(* IEC 61131-3 sources: TIA2AX/tests/V19/test_projects/expected/HW_2200330/ST50_PLC, 7 files *)

(* ---- HwIdentifiers.st ---- *)
TYPE
	HwIdentifiers : WORD
	(
		ST50_PLC_Profilschiene_0 :=	WORD#256,
		ST50_PLC :=	WORD#48,
		ST50_PLC_Card_reader_writer_1 :=	WORD#51,
		ST50_PLC_CPU_display_1 :=	WORD#54,
		ST50_PLC_OPC_UA_1 :=	WORD#117,
		ST50_PLC_DP_interface_1 :=	WORD#60,
		ST50_PLC_PROFINET_interface_1 :=	WORD#64,
		ST50_PLC_PROFINET_interface_1_Port_1 :=	WORD#65,
		ST50_PLC_PROFINET_interface_1_Port_2 :=	WORD#66,
		ST50_PLC_PROFINET_interface_2 :=	WORD#72,
		ST50_PLC_PROFINET_interface_2_Port_1 :=	WORD#73,
		ST50_Switch_SCALANCE_X_rack :=	WORD#393,
		ST50_Switch :=	WORD#394,
		ST50_Switch_ST50_Switch :=	WORD#395,
		ST50_Switch_SCALANCE_interface_1 :=	WORD#396,
		ST50_Switch_SCALANCE_interface_1_Port_1 :=	WORD#397,
		ST50_Switch_SCALANCE_interface_1_Port_2 :=	WORD#398,
		ST50_Switch_SCALANCE_interface_1_Port_3 :=	WORD#399,
		ST50_Switch_SCALANCE_interface_1_Port_4 :=	WORD#400,
		ST50_Switch_SCALANCE_interface_1_Port_5 :=	WORD#401,
		ST50_Switch_SCALANCE_interface_1_Port_6 :=	WORD#402,
		ST50_Switch_SCALANCE_interface_1_Port_7 :=	WORD#403,
		ST50_Switch_SCALANCE_interface_1_Port_8 :=	WORD#404,
		ST50_Switch_SCALANCE_interface_1_Port_9 :=	WORD#405,
		ST50_Switch_SCALANCE_interface_1_Port_10 :=	WORD#406,
		ST50_Switch_SCALANCE_interface_1_Port_11 :=	WORD#407,
		ST50_Switch_SCALANCE_interface_1_Port_12 :=	WORD#408,
		ST50_Switch_SCALANCE_interface_1_Port_13 :=	WORD#409,
		ST50_Switch_SCALANCE_interface_1_Port_14 :=	WORD#410,
		ST50_Switch_SCALANCE_interface_1_Port_15 :=	WORD#411,
		ST50_Switch_SCALANCE_interface_1_Port_16 :=	WORD#412,
		ST50_Switch_1_SCALANCE_X_rack :=	WORD#416,
		ST50_Switch_1 :=	WORD#417,
		ST50_Switch_1_ST50_Switch_1 :=	WORD#418,
		ST50_Switch_1_SCALANCE_interface_1 :=	WORD#419,
		ST50_Switch_1_SCALANCE_interface_1_Port_1 :=	WORD#420,
		ST50_Switch_1_SCALANCE_interface_1_Port_2 :=	WORD#421,
		ST50_Switch_1_SCALANCE_interface_1_Port_3 :=	WORD#422,
		ST50_Switch_1_SCALANCE_interface_1_Port_4 :=	WORD#423,
		ST50_Switch_1_SCALANCE_interface_1_Port_5 :=	WORD#424,
		ST50_Switch_1_SCALANCE_interface_1_Port_6 :=	WORD#425,
		ST50_Switch_1_SCALANCE_interface_1_Port_7 :=	WORD#426,
		ST50_Switch_1_SCALANCE_interface_1_Port_8 :=	WORD#427,
		ST50_Switch_1_SCALANCE_interface_1_Port_9 :=	WORD#428,
		ST50_Switch_1_SCALANCE_interface_1_Port_10 :=	WORD#429,
		ST50_Switch_1_SCALANCE_interface_1_Port_11 :=	WORD#430,
		ST50_Switch_1_SCALANCE_interface_1_Port_12 :=	WORD#431,
		ST50_Switch_1_SCALANCE_interface_1_Port_13 :=	WORD#432,
		ST50_Switch_1_SCALANCE_interface_1_Port_14 :=	WORD#433,
		ST50_Switch_1_SCALANCE_interface_1_Port_15 :=	WORD#434,
		ST50_Switch_1_SCALANCE_interface_1_Port_16 :=	WORD#435,
		ST50_CPX_PN_IO_Interface :=	WORD#259,
		ST50_CPX_PN_IO_Interface_Port_1 :=	WORD#260,
		ST50_CPX_PN_IO_Interface_Port_2 :=	WORD#261,
		ST50_CPX_CPX :=	WORD#262,
		ST50_CPX_MPA1S_VMPA1_FB_EMS_8_8DO_1 :=	WORD#263,
		ST50_CPX_MPA1S_VMPA1_FB_EMS_8_8DO_2 :=	WORD#264,
		ST50_CPX_MPA1S_VMPA1_FB_EMS_8_8DO_3 :=	WORD#265,
		ST50_CPX_MPA1S_VMPA1_FB_EMS_8_8DO_4 :=	WORD#266,
		ST50_CPX_MPA1S_VMPA1_FB_EMS_8_8DO_5 :=	WORD#267,
		ST50_CPX_MPA1S_VMPA1_FB_EMS_8_8DO_6 :=	WORD#268,
		ST50_CPX_MPA1S_VMPA1_FB_EMS_8_8DO_7 :=	WORD#269,
		ST50_CPX_MPA1S_VMPA1_FB_EMS_8_8DO_8 :=	WORD#270,
		ST50_CPX_MPA1S_VMPA1_FB_EMS_8_8DO_9 :=	WORD#271,
		ST50_CPX_MPA1G_VMPA1_FB_EMG_8_8DO_6 :=	WORD#272,
		ST50_ET200SP_Rack_0 :=	WORD#277,
		ST50_ET200SP :=	WORD#278,
		ST50_ET200SP_ST50_ET200SP :=	WORD#279,
		ST50_ET200SP_PROFINET_interface :=	WORD#280,
		ST50_ET200SP_PROFINET_interface_Port_1 :=	WORD#282,
		ST50_ET200SP_PROFINET_interface_Port_2 :=	WORD#281,
		ST50_ET200SP_BA_2xRJ45 :=	WORD#282,
		ST50_ET200SP_CM_4xIO_Link_1 :=	WORD#283,
		ST50_ET200SP_CM_4xIO_Link_2 :=	WORD#284,
		ST50_ET200SP_DI_16x24VDC_ST_1 :=	WORD#285,
		ST50_ET200SP_DI_16x24VDC_ST_2 :=	WORD#286,
		ST50_ET200SP_DI_8x24VDC_ST_4 :=	WORD#287,
		ST50_ET200SP_DI_8x24VDC_ST_3 :=	WORD#288,
		ST50_ET200SP_DQ_16x24VDC_0_5A_ST_1 :=	WORD#289,
		ST50_ET200SP_DQ_16x24VDC_0_5A_ST_2 :=	WORD#290,
		ST50_ET200SP_DQ_16x24VDC_0_5A_ST_3 :=	WORD#291,
		ST50_ET200SP_Servermodul_1 :=	WORD#292,
		ST50_HMI_ConnectionBox_Connection_Box :=	WORD#294,
		ST50_HMI_ConnectionBox :=	WORD#295,
		ST50_HMI_ConnectionBox_ST50_HMI_ConnectionBox :=	WORD#296,
		ST50_HMI_ConnectionBox_SCALANCE_interface_1 :=	WORD#297,
		ST50_HMI_ConnectionBox_SCALANCE_interface_1_Port_1 :=	WORD#298,
		ST50_HMI_ConnectionBox_SCALANCE_interface_1_Port_2 :=	WORD#299,
		ST50_HMI_ConnectionBox_SCALANCE_interface_1_Port_3 :=	WORD#300,
		ST50_SCHUNK_L_Rack :=	WORD#302,
		ST50_SCHUNK_L :=	WORD#303,
		ST50_SCHUNK_L_Interface :=	WORD#304,
		ST50_SCHUNK_L_Interface_Port_1 :=	WORD#305,
		ST50_SCHUNK_L_Interface_Port_2 :=	WORD#306,
		ST50_SCHUNK_L_DEVICE_SFP :=	WORD#307,
		ST50_SCHUNK_L_IN_4_Double_Words :=	WORD#308,
		ST50_SCHUNK_L_OUT_4_Double_Words :=	WORD#309,
		ST50_SCHUNK_R_Rack :=	WORD#311,
		ST50_SCHUNK_R :=	WORD#312,
		ST50_SCHUNK_R_Interface :=	WORD#313,
		ST50_SCHUNK_R_Interface_Port_1 :=	WORD#314,
		ST50_SCHUNK_R_Interface_Port_2 :=	WORD#315,
		ST50_SCHUNK_R_DEVICE_SFP :=	WORD#316,
		ST50_SCHUNK_R_IN_4_Double_Words :=	WORD#317,
		ST50_SCHUNK_R_OUT_4_Double_Words :=	WORD#318,
		ST50_TZ535_PN_Rack :=	WORD#320,
		ST50_TZ535_PN :=	WORD#321,
		ST50_TZ535_PN_Interface :=	WORD#322,
		ST50_TZ535_PN_Interface_Port_1 :=	WORD#323,
		ST50_TZ535_PN_Interface_Port_2 :=	WORD#324,
		ST50_TZ535_PN_2D_TZ535_PN_PROFINET_IO :=	WORD#325,
		ST50_TZ535_PN_In_Out_32_byte_x :=	WORD#326,
		ST50_1_DM260_WPC_Rack :=	WORD#328,
		ST50_1_DM260_WPC :=	WORD#329,
		ST50_1_DM260_WPC_Interface :=	WORD#330,
		ST50_1_DM260_WPC_Interface_Port_1 :=	WORD#331,
		ST50_1_DM260_WPC_DataMan_260 :=	WORD#332,
		ST50_1_DM260_WPC_Acquisition_Control :=	WORD#333,
		ST50_1_DM260_WPC_Acquisition_Status :=	WORD#334,
		ST50_1_DM260_WPC_Results_Control :=	WORD#335,
		ST50_1_DM260_WPC_Results_Status :=	WORD#336,
		ST50_1_DM260_WPC_Soft_Event_Control :=	WORD#337,
		ST50_1_DM260_WPC_User_Data_64_bytes :=	WORD#338,
		ST50_1_DM260_WPC_Result_Data_64_bytes :=	WORD#339,
		ST50_1_DM260_Rack :=	WORD#341,
		ST50_1_DM260 :=	WORD#342,
		ST50_1_DM260_Interface :=	WORD#343,
		ST50_1_DM260_Interface_Port_1 :=	WORD#344,
		ST50_1_DM260_DataMan_260 :=	WORD#345,
		ST50_1_DM260_Acquisition_Control :=	WORD#346,
		ST50_1_DM260_Acquisition_Status :=	WORD#347,
		ST50_1_DM260_Results_Control :=	WORD#348,
		ST50_1_DM260_Results_Status :=	WORD#349,
		ST50_1_DM260_Soft_Event_Control :=	WORD#350,
		ST50_1_DM260_User_Data_64_bytes :=	WORD#351,
		ST50_1_DM260_Result_Data_64_bytes :=	WORD#352,
		ST50_2_DM260_Rack :=	WORD#354,
		ST50_2_DM260 :=	WORD#355,
		ST50_2_DM260_Interface :=	WORD#356,
		ST50_2_DM260_Interface_Port_1 :=	WORD#357,
		ST50_2_DM260_DataMan_260 :=	WORD#358,
		ST50_2_DM260_Acquisition_Control :=	WORD#359,
		ST50_2_DM260_Acquisition_Status :=	WORD#360,
		ST50_2_DM260_Results_Control :=	WORD#361,
		ST50_2_DM260_Results_Status :=	WORD#362,
		ST50_2_DM260_Soft_Event_Control :=	WORD#363,
		ST50_2_DM260_User_Data_64_bytes :=	WORD#364,
		ST50_2_DM260_Result_Data_64_bytes :=	WORD#365,
		ST50_3_DM260_Rack :=	WORD#367,
		ST50_3_DM260 :=	WORD#368,
		ST50_3_DM260_Interface :=	WORD#369,
		ST50_3_DM260_Interface_Port_1 :=	WORD#370,
		ST50_3_DM260_DataMan_260 :=	WORD#371,
		ST50_3_DM260_Acquisition_Control :=	WORD#372,
		ST50_3_DM260_Acquisition_Status :=	WORD#373,
		ST50_3_DM260_Results_Control :=	WORD#374,
		ST50_3_DM260_Results_Status :=	WORD#375,
		ST50_3_DM260_Soft_Event_Control :=	WORD#376,
		ST50_3_DM260_User_Data_64_bytes :=	WORD#377,
		ST50_3_DM260_Result_Data_64_bytes :=	WORD#378,
		ST50_4_DM260_Rack :=	WORD#380,
		ST50_4_DM260 :=	WORD#381,
		ST50_4_DM260_Interface :=	WORD#382,
		ST50_4_DM260_Interface_Port_1 :=	WORD#383,
		ST50_4_DM260_DataMan_260 :=	WORD#384,
		ST50_4_DM260_Acquisition_Control :=	WORD#385,
		ST50_4_DM260_Acquisition_Status :=	WORD#386,
		ST50_4_DM260_Results_Control :=	WORD#387,
		ST50_4_DM260_Results_Status :=	WORD#388,
		ST50_4_DM260_Soft_Event_Control :=	WORD#389,
		ST50_4_DM260_User_Data_64_bytes :=	WORD#390,
		ST50_4_DM260_Result_Data_64_bytes :=	WORD#391,
		NONE:= WORD#0
	);
END_TYPE

(* ---- HwInputs.st ---- *)
TYPE
	HwInputs : STRUCT
		ST50_ET200SP_CM_4xIO_Link_1 AT %B100 : ARRAY[0..31] OF BYTE;
		ST50_ET200SP_CM_4xIO_Link_2 AT %B132 : ARRAY[0..31] OF BYTE;
		ST50_ET200SP_DI_16x24VDC_ST_1 AT %B0 : WORD;
		ST50_ET200SP_DI_16x24VDC_ST_2 AT %B2 : WORD;
		ST50_ET200SP_DI_8x24VDC_ST_4 AT %B4 : BYTE;
		ST50_ET200SP_DI_8x24VDC_ST_3 AT %B5 : BYTE;
		ST50_SCHUNK_L_IN_4_Double_Words AT %B600 : ARRAY[0..15] OF BYTE;
		ST50_SCHUNK_R_IN_4_Double_Words AT %B616 : ARRAY[0..15] OF BYTE;
		ST50_TZ535_PN_In_Out_32_byte_x AT %B1000 : ARRAY[0..31] OF BYTE;
		ST50_1_DM260_WPC_Acquisition_Status AT %B3505 : ARRAY[0..2] OF BYTE;
		ST50_1_DM260_WPC_Results_Status AT %B3508 : BYTE;
		ST50_1_DM260_WPC_Soft_Event_Control AT %B3509 : BYTE;
		ST50_1_DM260_WPC_Result_Data_64_bytes AT %B3582 : ARRAY[0..71] OF BYTE;
		ST50_1_DM260_Acquisition_Status AT %B3654 : ARRAY[0..2] OF BYTE;
		ST50_1_DM260_Results_Status AT %B3657 : BYTE;
		ST50_1_DM260_Soft_Event_Control AT %B3658 : BYTE;
		ST50_1_DM260_Result_Data_64_bytes AT %B3659 : ARRAY[0..71] OF BYTE;
		ST50_2_DM260_Acquisition_Status AT %B3731 : ARRAY[0..2] OF BYTE;
		ST50_2_DM260_Results_Status AT %B3734 : BYTE;
		ST50_2_DM260_Soft_Event_Control AT %B3735 : BYTE;
		ST50_2_DM260_Result_Data_64_bytes AT %B3736 : ARRAY[0..71] OF BYTE;
		ST50_3_DM260_Acquisition_Status AT %B3808 : ARRAY[0..2] OF BYTE;
		ST50_3_DM260_Results_Status AT %B3811 : BYTE;
		ST50_3_DM260_Soft_Event_Control AT %B3812 : BYTE;
		ST50_3_DM260_Result_Data_64_bytes AT %B3813 : ARRAY[0..71] OF BYTE;
		ST50_4_DM260_Acquisition_Status AT %B3885 : ARRAY[0..2] OF BYTE;
		ST50_4_DM260_Results_Status AT %B3888 : BYTE;
		ST50_4_DM260_Soft_Event_Control AT %B3889 : BYTE;
		ST50_4_DM260_Result_Data_64_bytes AT %B3890 : ARRAY[0..71] OF BYTE;
	END_STRUCT;
END_TYPE

(* ---- HwOutputs.st ---- *)
TYPE
	HwOutputs : STRUCT
		ST50_CPX_MPA1S_VMPA1_FB_EMS_8_8DO_1 AT %B200 : BYTE;
		ST50_CPX_MPA1S_VMPA1_FB_EMS_8_8DO_2 AT %B201 : BYTE;
		ST50_CPX_MPA1S_VMPA1_FB_EMS_8_8DO_3 AT %B202 : BYTE;
		ST50_CPX_MPA1S_VMPA1_FB_EMS_8_8DO_4 AT %B203 : BYTE;
		ST50_CPX_MPA1S_VMPA1_FB_EMS_8_8DO_5 AT %B204 : BYTE;
		ST50_CPX_MPA1S_VMPA1_FB_EMS_8_8DO_6 AT %B205 : BYTE;
		ST50_CPX_MPA1S_VMPA1_FB_EMS_8_8DO_7 AT %B206 : BYTE;
		ST50_CPX_MPA1S_VMPA1_FB_EMS_8_8DO_8 AT %B207 : BYTE;
		ST50_CPX_MPA1S_VMPA1_FB_EMS_8_8DO_9 AT %B208 : BYTE;
		ST50_CPX_MPA1G_VMPA1_FB_EMG_8_8DO_6 AT %B209 : BYTE;
		ST50_ET200SP_CM_4xIO_Link_1 AT %B100 : ARRAY[0..31] OF BYTE;
		ST50_ET200SP_CM_4xIO_Link_2 AT %B132 : ARRAY[0..31] OF BYTE;
		ST50_ET200SP_DQ_16x24VDC_0_5A_ST_1 AT %B0 : WORD;
		ST50_ET200SP_DQ_16x24VDC_0_5A_ST_2 AT %B2 : WORD;
		ST50_ET200SP_DQ_16x24VDC_0_5A_ST_3 AT %B4 : WORD;
		ST50_SCHUNK_L_OUT_4_Double_Words AT %B600 : ARRAY[0..15] OF BYTE;
		ST50_SCHUNK_R_OUT_4_Double_Words AT %B616 : ARRAY[0..15] OF BYTE;
		ST50_TZ535_PN_In_Out_32_byte_x AT %B1000 : ARRAY[0..31] OF BYTE;
		ST50_1_DM260_WPC_Acquisition_Control AT %B3501 : BYTE;
		ST50_1_DM260_WPC_Results_Control AT %B3505 : BYTE;
		ST50_1_DM260_WPC_Soft_Event_Control AT %B3506 : BYTE;
		ST50_1_DM260_WPC_User_Data_64_bytes AT %B3578 : ARRAY[0..67] OF BYTE;
		ST50_1_DM260_Acquisition_Control AT %B3502 : BYTE;
		ST50_1_DM260_Results_Control AT %B3507 : BYTE;
		ST50_1_DM260_Soft_Event_Control AT %B3508 : BYTE;
		ST50_1_DM260_User_Data_64_bytes AT %B3646 : ARRAY[0..67] OF BYTE;
		ST50_2_DM260_Acquisition_Control AT %B3509 : BYTE;
		ST50_2_DM260_Results_Control AT %B3714 : BYTE;
		ST50_2_DM260_Soft_Event_Control AT %B3715 : BYTE;
		ST50_2_DM260_User_Data_64_bytes AT %B3716 : ARRAY[0..67] OF BYTE;
		ST50_3_DM260_Acquisition_Control AT %B3784 : BYTE;
		ST50_3_DM260_Results_Control AT %B3785 : BYTE;
		ST50_3_DM260_Soft_Event_Control AT %B3786 : BYTE;
		ST50_3_DM260_User_Data_64_bytes AT %B3787 : ARRAY[0..67] OF BYTE;
		ST50_4_DM260_Acquisition_Control AT %B3855 : BYTE;
		ST50_4_DM260_Results_Control AT %B3856 : BYTE;
		ST50_4_DM260_Soft_Event_Control AT %B3857 : BYTE;
		ST50_4_DM260_User_Data_64_bytes AT %B3858 : ARRAY[0..67] OF BYTE;
	END_STRUCT;
END_TYPE

(* ---- PlcInputs.st ---- *)
TYPE
	PlcInputs : STRUCT
		ST50_ET200SP_CM_4xIO_Link_1 : ARRAY[0..31] OF BYTE;
		ST50_ET200SP_CM_4xIO_Link_2 : ARRAY[0..31] OF BYTE;
		ST50_ET200SP_DI_16x24VDC_ST_1 : WORD;
		ST50_ET200SP_DI_16x24VDC_ST_2 : WORD;
		ST50_ET200SP_DI_8x24VDC_ST_4 : BYTE;
		ST50_ET200SP_DI_8x24VDC_ST_3 : BYTE;
		ST50_SCHUNK_L_IN_4_Double_Words : ARRAY[0..15] OF BYTE;
		ST50_SCHUNK_R_IN_4_Double_Words : ARRAY[0..15] OF BYTE;
		ST50_TZ535_PN_In_Out_32_byte_x : ARRAY[0..31] OF BYTE;
		ST50_1_DM260_WPC_Acquisition_Status : ARRAY[0..2] OF BYTE;
		ST50_1_DM260_WPC_Results_Status : BYTE;
		ST50_1_DM260_WPC_Soft_Event_Control : BYTE;
		ST50_1_DM260_WPC_Result_Data_64_bytes : ARRAY[0..71] OF BYTE;
		ST50_1_DM260_Acquisition_Status : ARRAY[0..2] OF BYTE;
		ST50_1_DM260_Results_Status : BYTE;
		ST50_1_DM260_Soft_Event_Control : BYTE;
		ST50_1_DM260_Result_Data_64_bytes : ARRAY[0..71] OF BYTE;
		ST50_2_DM260_Acquisition_Status : ARRAY[0..2] OF BYTE;
		ST50_2_DM260_Results_Status : BYTE;
		ST50_2_DM260_Soft_Event_Control : BYTE;
		ST50_2_DM260_Result_Data_64_bytes : ARRAY[0..71] OF BYTE;
		ST50_3_DM260_Acquisition_Status : ARRAY[0..2] OF BYTE;
		ST50_3_DM260_Results_Status : BYTE;
		ST50_3_DM260_Soft_Event_Control : BYTE;
		ST50_3_DM260_Result_Data_64_bytes : ARRAY[0..71] OF BYTE;
		ST50_4_DM260_Acquisition_Status : ARRAY[0..2] OF BYTE;
		ST50_4_DM260_Results_Status : BYTE;
		ST50_4_DM260_Soft_Event_Control : BYTE;
		ST50_4_DM260_Result_Data_64_bytes : ARRAY[0..71] OF BYTE;
	END_STRUCT;
END_TYPE

(* ---- PlcOutputs.st ---- *)
TYPE
	PlcOutputs : STRUCT
		ST50_CPX_MPA1S_VMPA1_FB_EMS_8_8DO_1 : BYTE;
		ST50_CPX_MPA1S_VMPA1_FB_EMS_8_8DO_2 : BYTE;
		ST50_CPX_MPA1S_VMPA1_FB_EMS_8_8DO_3 : BYTE;
		ST50_CPX_MPA1S_VMPA1_FB_EMS_8_8DO_4 : BYTE;
		ST50_CPX_MPA1S_VMPA1_FB_EMS_8_8DO_5 : BYTE;
		ST50_CPX_MPA1S_VMPA1_FB_EMS_8_8DO_6 : BYTE;
		ST50_CPX_MPA1S_VMPA1_FB_EMS_8_8DO_7 : BYTE;
		ST50_CPX_MPA1S_VMPA1_FB_EMS_8_8DO_8 : BYTE;
		ST50_CPX_MPA1S_VMPA1_FB_EMS_8_8DO_9 : BYTE;
		ST50_CPX_MPA1G_VMPA1_FB_EMG_8_8DO_6 : BYTE;
		ST50_ET200SP_CM_4xIO_Link_1 : ARRAY[0..31] OF BYTE;
		ST50_ET200SP_CM_4xIO_Link_2 : ARRAY[0..31] OF BYTE;
		ST50_ET200SP_DQ_16x24VDC_0_5A_ST_1 : WORD;
		ST50_ET200SP_DQ_16x24VDC_0_5A_ST_2 : WORD;
		ST50_ET200SP_DQ_16x24VDC_0_5A_ST_3 : WORD;
		ST50_SCHUNK_L_OUT_4_Double_Words : ARRAY[0..15] OF BYTE;
		ST50_SCHUNK_R_OUT_4_Double_Words : ARRAY[0..15] OF BYTE;
		ST50_TZ535_PN_In_Out_32_byte_x : ARRAY[0..31] OF BYTE;
		ST50_1_DM260_WPC_Acquisition_Control : BYTE;
		ST50_1_DM260_WPC_Results_Control : BYTE;
		ST50_1_DM260_WPC_Soft_Event_Control : BYTE;
		ST50_1_DM260_WPC_User_Data_64_bytes : ARRAY[0..67] OF BYTE;
		ST50_1_DM260_Acquisition_Control : BYTE;
		ST50_1_DM260_Results_Control : BYTE;
		ST50_1_DM260_Soft_Event_Control : BYTE;
		ST50_1_DM260_User_Data_64_bytes : ARRAY[0..67] OF BYTE;
		ST50_2_DM260_Acquisition_Control : BYTE;
		ST50_2_DM260_Results_Control : BYTE;
		ST50_2_DM260_Soft_Event_Control : BYTE;
		ST50_2_DM260_User_Data_64_bytes : ARRAY[0..67] OF BYTE;
		ST50_3_DM260_Acquisition_Control : BYTE;
		ST50_3_DM260_Results_Control : BYTE;
		ST50_3_DM260_Soft_Event_Control : BYTE;
		ST50_3_DM260_User_Data_64_bytes : ARRAY[0..67] OF BYTE;
		ST50_4_DM260_Acquisition_Control : BYTE;
		ST50_4_DM260_Results_Control : BYTE;
		ST50_4_DM260_Soft_Event_Control : BYTE;
		ST50_4_DM260_User_Data_64_bytes : ARRAY[0..67] OF BYTE;
	END_STRUCT;
END_TYPE

(* ---- CopyInputs.st ---- *)
FUNCTION CopyInputs
	VAR_EXTERNAL
		HwInputs : HwInputs;
		PlcInputs : PlcInputs;
	END_VAR
	PlcInputs.ST50_ET200SP_CM_4xIO_Link_1[0] := HwInputs.ST50_ET200SP_CM_4xIO_Link_1[0];
	PlcInputs.ST50_ET200SP_CM_4xIO_Link_1[1] := HwInputs.ST50_ET200SP_CM_4xIO_Link_1[1];
	PlcInputs.ST50_ET200SP_CM_4xIO_Link_1[2] := HwInputs.ST50_ET200SP_CM_4xIO_Link_1[2];
	PlcInputs.ST50_ET200SP_CM_4xIO_Link_1[3] := HwInputs.ST50_ET200SP_CM_4xIO_Link_1[3];
	PlcInputs.ST50_ET200SP_CM_4xIO_Link_1[4] := HwInputs.ST50_ET200SP_CM_4xIO_Link_1[4];
	PlcInputs.ST50_ET200SP_CM_4xIO_Link_1[5] := HwInputs.ST50_ET200SP_CM_4xIO_Link_1[5];
	PlcInputs.ST50_ET200SP_CM_4xIO_Link_1[6] := HwInputs.ST50_ET200SP_CM_4xIO_Link_1[6];
	PlcInputs.ST50_ET200SP_CM_4xIO_Link_1[7] := HwInputs.ST50_ET200SP_CM_4xIO_Link_1[7];
	PlcInputs.ST50_ET200SP_CM_4xIO_Link_1[8] := HwInputs.ST50_ET200SP_CM_4xIO_Link_1[8];
	PlcInputs.ST50_ET200SP_CM_4xIO_Link_1[9] := HwInputs.ST50_ET200SP_CM_4xIO_Link_1[9];
	PlcInputs.ST50_ET200SP_CM_4xIO_Link_1[10] := HwInputs.ST50_ET200SP_CM_4xIO_Link_1[10];
	PlcInputs.ST50_ET200SP_CM_4xIO_Link_1[11] := HwInputs.ST50_ET200SP_CM_4xIO_Link_1[11];
	PlcInputs.ST50_ET200SP_CM_4xIO_Link_1[12] := HwInputs.ST50_ET200SP_CM_4xIO_Link_1[12];
	PlcInputs.ST50_ET200SP_CM_4xIO_Link_1[13] := HwInputs.ST50_ET200SP_CM_4xIO_Link_1[13];
	PlcInputs.ST50_ET200SP_CM_4xIO_Link_1[14] := HwInputs.ST50_ET200SP_CM_4xIO_Link_1[14];
	PlcInputs.ST50_ET200SP_CM_4xIO_Link_1[15] := HwInputs.ST50_ET200SP_CM_4xIO_Link_1[15];
	PlcInputs.ST50_ET200SP_CM_4xIO_Link_1[16] := HwInputs.ST50_ET200SP_CM_4xIO_Link_1[16];
	PlcInputs.ST50_ET200SP_CM_4xIO_Link_1[17] := HwInputs.ST50_ET200SP_CM_4xIO_Link_1[17];
	PlcInputs.ST50_ET200SP_CM_4xIO_Link_1[18] := HwInputs.ST50_ET200SP_CM_4xIO_Link_1[18];
	PlcInputs.ST50_ET200SP_CM_4xIO_Link_1[19] := HwInputs.ST50_ET200SP_CM_4xIO_Link_1[19];
	PlcInputs.ST50_ET200SP_CM_4xIO_Link_1[20] := HwInputs.ST50_ET200SP_CM_4xIO_Link_1[20];
	PlcInputs.ST50_ET200SP_CM_4xIO_Link_1[21] := HwInputs.ST50_ET200SP_CM_4xIO_Link_1[21];
	PlcInputs.ST50_ET200SP_CM_4xIO_Link_1[22] := HwInputs.ST50_ET200SP_CM_4xIO_Link_1[22];
	PlcInputs.ST50_ET200SP_CM_4xIO_Link_1[23] := HwInputs.ST50_ET200SP_CM_4xIO_Link_1[23];
	PlcInputs.ST50_ET200SP_CM_4xIO_Link_1[24] := HwInputs.ST50_ET200SP_CM_4xIO_Link_1[24];
	PlcInputs.ST50_ET200SP_CM_4xIO_Link_1[25] := HwInputs.ST50_ET200SP_CM_4xIO_Link_1[25];
	PlcInputs.ST50_ET200SP_CM_4xIO_Link_1[26] := HwInputs.ST50_ET200SP_CM_4xIO_Link_1[26];
	PlcInputs.ST50_ET200SP_CM_4xIO_Link_1[27] := HwInputs.ST50_ET200SP_CM_4xIO_Link_1[27];
	PlcInputs.ST50_ET200SP_CM_4xIO_Link_1[28] := HwInputs.ST50_ET200SP_CM_4xIO_Link_1[28];
	PlcInputs.ST50_ET200SP_CM_4xIO_Link_1[29] := HwInputs.ST50_ET200SP_CM_4xIO_Link_1[29];
	PlcInputs.ST50_ET200SP_CM_4xIO_Link_1[30] := HwInputs.ST50_ET200SP_CM_4xIO_Link_1[30];
	PlcInputs.ST50_ET200SP_CM_4xIO_Link_1[31] := HwInputs.ST50_ET200SP_CM_4xIO_Link_1[31];
	PlcInputs.ST50_ET200SP_CM_4xIO_Link_2[0] := HwInputs.ST50_ET200SP_CM_4xIO_Link_2[0];
	PlcInputs.ST50_ET200SP_CM_4xIO_Link_2[1] := HwInputs.ST50_ET200SP_CM_4xIO_Link_2[1];
	PlcInputs.ST50_ET200SP_CM_4xIO_Link_2[2] := HwInputs.ST50_ET200SP_CM_4xIO_Link_2[2];
	PlcInputs.ST50_ET200SP_CM_4xIO_Link_2[3] := HwInputs.ST50_ET200SP_CM_4xIO_Link_2[3];
	PlcInputs.ST50_ET200SP_CM_4xIO_Link_2[4] := HwInputs.ST50_ET200SP_CM_4xIO_Link_2[4];
	PlcInputs.ST50_ET200SP_CM_4xIO_Link_2[5] := HwInputs.ST50_ET200SP_CM_4xIO_Link_2[5];
	PlcInputs.ST50_ET200SP_CM_4xIO_Link_2[6] := HwInputs.ST50_ET200SP_CM_4xIO_Link_2[6];
	PlcInputs.ST50_ET200SP_CM_4xIO_Link_2[7] := HwInputs.ST50_ET200SP_CM_4xIO_Link_2[7];
	PlcInputs.ST50_ET200SP_CM_4xIO_Link_2[8] := HwInputs.ST50_ET200SP_CM_4xIO_Link_2[8];
	PlcInputs.ST50_ET200SP_CM_4xIO_Link_2[9] := HwInputs.ST50_ET200SP_CM_4xIO_Link_2[9];
	PlcInputs.ST50_ET200SP_CM_4xIO_Link_2[10] := HwInputs.ST50_ET200SP_CM_4xIO_Link_2[10];
	PlcInputs.ST50_ET200SP_CM_4xIO_Link_2[11] := HwInputs.ST50_ET200SP_CM_4xIO_Link_2[11];
	PlcInputs.ST50_ET200SP_CM_4xIO_Link_2[12] := HwInputs.ST50_ET200SP_CM_4xIO_Link_2[12];
	PlcInputs.ST50_ET200SP_CM_4xIO_Link_2[13] := HwInputs.ST50_ET200SP_CM_4xIO_Link_2[13];
	PlcInputs.ST50_ET200SP_CM_4xIO_Link_2[14] := HwInputs.ST50_ET200SP_CM_4xIO_Link_2[14];
	PlcInputs.ST50_ET200SP_CM_4xIO_Link_2[15] := HwInputs.ST50_ET200SP_CM_4xIO_Link_2[15];
	PlcInputs.ST50_ET200SP_CM_4xIO_Link_2[16] := HwInputs.ST50_ET200SP_CM_4xIO_Link_2[16];
	PlcInputs.ST50_ET200SP_CM_4xIO_Link_2[17] := HwInputs.ST50_ET200SP_CM_4xIO_Link_2[17];
	PlcInputs.ST50_ET200SP_CM_4xIO_Link_2[18] := HwInputs.ST50_ET200SP_CM_4xIO_Link_2[18];
	PlcInputs.ST50_ET200SP_CM_4xIO_Link_2[19] := HwInputs.ST50_ET200SP_CM_4xIO_Link_2[19];
	PlcInputs.ST50_ET200SP_CM_4xIO_Link_2[20] := HwInputs.ST50_ET200SP_CM_4xIO_Link_2[20];
	PlcInputs.ST50_ET200SP_CM_4xIO_Link_2[21] := HwInputs.ST50_ET200SP_CM_4xIO_Link_2[21];
	PlcInputs.ST50_ET200SP_CM_4xIO_Link_2[22] := HwInputs.ST50_ET200SP_CM_4xIO_Link_2[22];
	PlcInputs.ST50_ET200SP_CM_4xIO_Link_2[23] := HwInputs.ST50_ET200SP_CM_4xIO_Link_2[23];
	PlcInputs.ST50_ET200SP_CM_4xIO_Link_2[24] := HwInputs.ST50_ET200SP_CM_4xIO_Link_2[24];
	PlcInputs.ST50_ET200SP_CM_4xIO_Link_2[25] := HwInputs.ST50_ET200SP_CM_4xIO_Link_2[25];
	PlcInputs.ST50_ET200SP_CM_4xIO_Link_2[26] := HwInputs.ST50_ET200SP_CM_4xIO_Link_2[26];
	PlcInputs.ST50_ET200SP_CM_4xIO_Link_2[27] := HwInputs.ST50_ET200SP_CM_4xIO_Link_2[27];
	PlcInputs.ST50_ET200SP_CM_4xIO_Link_2[28] := HwInputs.ST50_ET200SP_CM_4xIO_Link_2[28];
	PlcInputs.ST50_ET200SP_CM_4xIO_Link_2[29] := HwInputs.ST50_ET200SP_CM_4xIO_Link_2[29];
	PlcInputs.ST50_ET200SP_CM_4xIO_Link_2[30] := HwInputs.ST50_ET200SP_CM_4xIO_Link_2[30];
	PlcInputs.ST50_ET200SP_CM_4xIO_Link_2[31] := HwInputs.ST50_ET200SP_CM_4xIO_Link_2[31];
	PlcInputs.ST50_ET200SP_DI_16x24VDC_ST_1 := HwInputs.ST50_ET200SP_DI_16x24VDC_ST_1;
	PlcInputs.ST50_ET200SP_DI_16x24VDC_ST_2 := HwInputs.ST50_ET200SP_DI_16x24VDC_ST_2;
	PlcInputs.ST50_ET200SP_DI_8x24VDC_ST_4 := HwInputs.ST50_ET200SP_DI_8x24VDC_ST_4;
	PlcInputs.ST50_ET200SP_DI_8x24VDC_ST_3 := HwInputs.ST50_ET200SP_DI_8x24VDC_ST_3;
	PlcInputs.ST50_SCHUNK_L_IN_4_Double_Words[0] := HwInputs.ST50_SCHUNK_L_IN_4_Double_Words[0];
	PlcInputs.ST50_SCHUNK_L_IN_4_Double_Words[1] := HwInputs.ST50_SCHUNK_L_IN_4_Double_Words[1];
	PlcInputs.ST50_SCHUNK_L_IN_4_Double_Words[2] := HwInputs.ST50_SCHUNK_L_IN_4_Double_Words[2];
	PlcInputs.ST50_SCHUNK_L_IN_4_Double_Words[3] := HwInputs.ST50_SCHUNK_L_IN_4_Double_Words[3];
	PlcInputs.ST50_SCHUNK_L_IN_4_Double_Words[4] := HwInputs.ST50_SCHUNK_L_IN_4_Double_Words[4];
	PlcInputs.ST50_SCHUNK_L_IN_4_Double_Words[5] := HwInputs.ST50_SCHUNK_L_IN_4_Double_Words[5];
	PlcInputs.ST50_SCHUNK_L_IN_4_Double_Words[6] := HwInputs.ST50_SCHUNK_L_IN_4_Double_Words[6];
	PlcInputs.ST50_SCHUNK_L_IN_4_Double_Words[7] := HwInputs.ST50_SCHUNK_L_IN_4_Double_Words[7];
	PlcInputs.ST50_SCHUNK_L_IN_4_Double_Words[8] := HwInputs.ST50_SCHUNK_L_IN_4_Double_Words[8];
	PlcInputs.ST50_SCHUNK_L_IN_4_Double_Words[9] := HwInputs.ST50_SCHUNK_L_IN_4_Double_Words[9];
	PlcInputs.ST50_SCHUNK_L_IN_4_Double_Words[10] := HwInputs.ST50_SCHUNK_L_IN_4_Double_Words[10];
	PlcInputs.ST50_SCHUNK_L_IN_4_Double_Words[11] := HwInputs.ST50_SCHUNK_L_IN_4_Double_Words[11];
	PlcInputs.ST50_SCHUNK_L_IN_4_Double_Words[12] := HwInputs.ST50_SCHUNK_L_IN_4_Double_Words[12];
	PlcInputs.ST50_SCHUNK_L_IN_4_Double_Words[13] := HwInputs.ST50_SCHUNK_L_IN_4_Double_Words[13];
	PlcInputs.ST50_SCHUNK_L_IN_4_Double_Words[14] := HwInputs.ST50_SCHUNK_L_IN_4_Double_Words[14];
	PlcInputs.ST50_SCHUNK_L_IN_4_Double_Words[15] := HwInputs.ST50_SCHUNK_L_IN_4_Double_Words[15];
	PlcInputs.ST50_SCHUNK_R_IN_4_Double_Words[0] := HwInputs.ST50_SCHUNK_R_IN_4_Double_Words[0];
	PlcInputs.ST50_SCHUNK_R_IN_4_Double_Words[1] := HwInputs.ST50_SCHUNK_R_IN_4_Double_Words[1];
	PlcInputs.ST50_SCHUNK_R_IN_4_Double_Words[2] := HwInputs.ST50_SCHUNK_R_IN_4_Double_Words[2];
	PlcInputs.ST50_SCHUNK_R_IN_4_Double_Words[3] := HwInputs.ST50_SCHUNK_R_IN_4_Double_Words[3];
	PlcInputs.ST50_SCHUNK_R_IN_4_Double_Words[4] := HwInputs.ST50_SCHUNK_R_IN_4_Double_Words[4];
	PlcInputs.ST50_SCHUNK_R_IN_4_Double_Words[5] := HwInputs.ST50_SCHUNK_R_IN_4_Double_Words[5];
	PlcInputs.ST50_SCHUNK_R_IN_4_Double_Words[6] := HwInputs.ST50_SCHUNK_R_IN_4_Double_Words[6];
	PlcInputs.ST50_SCHUNK_R_IN_4_Double_Words[7] := HwInputs.ST50_SCHUNK_R_IN_4_Double_Words[7];
	PlcInputs.ST50_SCHUNK_R_IN_4_Double_Words[8] := HwInputs.ST50_SCHUNK_R_IN_4_Double_Words[8];
	PlcInputs.ST50_SCHUNK_R_IN_4_Double_Words[9] := HwInputs.ST50_SCHUNK_R_IN_4_Double_Words[9];
	PlcInputs.ST50_SCHUNK_R_IN_4_Double_Words[10] := HwInputs.ST50_SCHUNK_R_IN_4_Double_Words[10];
	PlcInputs.ST50_SCHUNK_R_IN_4_Double_Words[11] := HwInputs.ST50_SCHUNK_R_IN_4_Double_Words[11];
	PlcInputs.ST50_SCHUNK_R_IN_4_Double_Words[12] := HwInputs.ST50_SCHUNK_R_IN_4_Double_Words[12];
	PlcInputs.ST50_SCHUNK_R_IN_4_Double_Words[13] := HwInputs.ST50_SCHUNK_R_IN_4_Double_Words[13];
	PlcInputs.ST50_SCHUNK_R_IN_4_Double_Words[14] := HwInputs.ST50_SCHUNK_R_IN_4_Double_Words[14];
	PlcInputs.ST50_SCHUNK_R_IN_4_Double_Words[15] := HwInputs.ST50_SCHUNK_R_IN_4_Double_Words[15];
	PlcInputs.ST50_TZ535_PN_In_Out_32_byte_x[0] := HwInputs.ST50_TZ535_PN_In_Out_32_byte_x[0];
	PlcInputs.ST50_TZ535_PN_In_Out_32_byte_x[1] := HwInputs.ST50_TZ535_PN_In_Out_32_byte_x[1];
	PlcInputs.ST50_TZ535_PN_In_Out_32_byte_x[2] := HwInputs.ST50_TZ535_PN_In_Out_32_byte_x[2];
	PlcInputs.ST50_TZ535_PN_In_Out_32_byte_x[3] := HwInputs.ST50_TZ535_PN_In_Out_32_byte_x[3];
	PlcInputs.ST50_TZ535_PN_In_Out_32_byte_x[4] := HwInputs.ST50_TZ535_PN_In_Out_32_byte_x[4];
	PlcInputs.ST50_TZ535_PN_In_Out_32_byte_x[5] := HwInputs.ST50_TZ535_PN_In_Out_32_byte_x[5];
	PlcInputs.ST50_TZ535_PN_In_Out_32_byte_x[6] := HwInputs.ST50_TZ535_PN_In_Out_32_byte_x[6];
	PlcInputs.ST50_TZ535_PN_In_Out_32_byte_x[7] := HwInputs.ST50_TZ535_PN_In_Out_32_byte_x[7];
	PlcInputs.ST50_TZ535_PN_In_Out_32_byte_x[8] := HwInputs.ST50_TZ535_PN_In_Out_32_byte_x[8];
	PlcInputs.ST50_TZ535_PN_In_Out_32_byte_x[9] := HwInputs.ST50_TZ535_PN_In_Out_32_byte_x[9];
	PlcInputs.ST50_TZ535_PN_In_Out_32_byte_x[10] := HwInputs.ST50_TZ535_PN_In_Out_32_byte_x[10];
	PlcInputs.ST50_TZ535_PN_In_Out_32_byte_x[11] := HwInputs.ST50_TZ535_PN_In_Out_32_byte_x[11];
	PlcInputs.ST50_TZ535_PN_In_Out_32_byte_x[12] := HwInputs.ST50_TZ535_PN_In_Out_32_byte_x[12];
	PlcInputs.ST50_TZ535_PN_In_Out_32_byte_x[13] := HwInputs.ST50_TZ535_PN_In_Out_32_byte_x[13];
	PlcInputs.ST50_TZ535_PN_In_Out_32_byte_x[14] := HwInputs.ST50_TZ535_PN_In_Out_32_byte_x[14];
	PlcInputs.ST50_TZ535_PN_In_Out_32_byte_x[15] := HwInputs.ST50_TZ535_PN_In_Out_32_byte_x[15];
	PlcInputs.ST50_TZ535_PN_In_Out_32_byte_x[16] := HwInputs.ST50_TZ535_PN_In_Out_32_byte_x[16];
	PlcInputs.ST50_TZ535_PN_In_Out_32_byte_x[17] := HwInputs.ST50_TZ535_PN_In_Out_32_byte_x[17];
	PlcInputs.ST50_TZ535_PN_In_Out_32_byte_x[18] := HwInputs.ST50_TZ535_PN_In_Out_32_byte_x[18];
	PlcInputs.ST50_TZ535_PN_In_Out_32_byte_x[19] := HwInputs.ST50_TZ535_PN_In_Out_32_byte_x[19];
	PlcInputs.ST50_TZ535_PN_In_Out_32_byte_x[20] := HwInputs.ST50_TZ535_PN_In_Out_32_byte_x[20];
	PlcInputs.ST50_TZ535_PN_In_Out_32_byte_x[21] := HwInputs.ST50_TZ535_PN_In_Out_32_byte_x[21];
	PlcInputs.ST50_TZ535_PN_In_Out_32_byte_x[22] := HwInputs.ST50_TZ535_PN_In_Out_32_byte_x[22];
	PlcInputs.ST50_TZ535_PN_In_Out_32_byte_x[23] := HwInputs.ST50_TZ535_PN_In_Out_32_byte_x[23];
	PlcInputs.ST50_TZ535_PN_In_Out_32_byte_x[24] := HwInputs.ST50_TZ535_PN_In_Out_32_byte_x[24];
	PlcInputs.ST50_TZ535_PN_In_Out_32_byte_x[25] := HwInputs.ST50_TZ535_PN_In_Out_32_byte_x[25];
	PlcInputs.ST50_TZ535_PN_In_Out_32_byte_x[26] := HwInputs.ST50_TZ535_PN_In_Out_32_byte_x[26];
	PlcInputs.ST50_TZ535_PN_In_Out_32_byte_x[27] := HwInputs.ST50_TZ535_PN_In_Out_32_byte_x[27];
	PlcInputs.ST50_TZ535_PN_In_Out_32_byte_x[28] := HwInputs.ST50_TZ535_PN_In_Out_32_byte_x[28];
	PlcInputs.ST50_TZ535_PN_In_Out_32_byte_x[29] := HwInputs.ST50_TZ535_PN_In_Out_32_byte_x[29];
	PlcInputs.ST50_TZ535_PN_In_Out_32_byte_x[30] := HwInputs.ST50_TZ535_PN_In_Out_32_byte_x[30];
	PlcInputs.ST50_TZ535_PN_In_Out_32_byte_x[31] := HwInputs.ST50_TZ535_PN_In_Out_32_byte_x[31];
	PlcInputs.ST50_1_DM260_WPC_Acquisition_Status[0] := HwInputs.ST50_1_DM260_WPC_Acquisition_Status[0];
	PlcInputs.ST50_1_DM260_WPC_Acquisition_Status[1] := HwInputs.ST50_1_DM260_WPC_Acquisition_Status[1];
	PlcInputs.ST50_1_DM260_WPC_Acquisition_Status[2] := HwInputs.ST50_1_DM260_WPC_Acquisition_Status[2];
	PlcInputs.ST50_1_DM260_WPC_Results_Status := HwInputs.ST50_1_DM260_WPC_Results_Status;
	PlcInputs.ST50_1_DM260_WPC_Soft_Event_Control := HwInputs.ST50_1_DM260_WPC_Soft_Event_Control;
	PlcInputs.ST50_1_DM260_WPC_Result_Data_64_bytes[0] := HwInputs.ST50_1_DM260_WPC_Result_Data_64_bytes[0];
	PlcInputs.ST50_1_DM260_WPC_Result_Data_64_bytes[1] := HwInputs.ST50_1_DM260_WPC_Result_Data_64_bytes[1];
	PlcInputs.ST50_1_DM260_WPC_Result_Data_64_bytes[2] := HwInputs.ST50_1_DM260_WPC_Result_Data_64_bytes[2];
	PlcInputs.ST50_1_DM260_WPC_Result_Data_64_bytes[3] := HwInputs.ST50_1_DM260_WPC_Result_Data_64_bytes[3];
	PlcInputs.ST50_1_DM260_WPC_Result_Data_64_bytes[4] := HwInputs.ST50_1_DM260_WPC_Result_Data_64_bytes[4];
	PlcInputs.ST50_1_DM260_WPC_Result_Data_64_bytes[5] := HwInputs.ST50_1_DM260_WPC_Result_Data_64_bytes[5];
	PlcInputs.ST50_1_DM260_WPC_Result_Data_64_bytes[6] := HwInputs.ST50_1_DM260_WPC_Result_Data_64_bytes[6];
	PlcInputs.ST50_1_DM260_WPC_Result_Data_64_bytes[7] := HwInputs.ST50_1_DM260_WPC_Result_Data_64_bytes[7];
	PlcInputs.ST50_1_DM260_WPC_Result_Data_64_bytes[8] := HwInputs.ST50_1_DM260_WPC_Result_Data_64_bytes[8];
	PlcInputs.ST50_1_DM260_WPC_Result_Data_64_bytes[9] := HwInputs.ST50_1_DM260_WPC_Result_Data_64_bytes[9];
	PlcInputs.ST50_1_DM260_WPC_Result_Data_64_bytes[10] := HwInputs.ST50_1_DM260_WPC_Result_Data_64_bytes[10];
	PlcInputs.ST50_1_DM260_WPC_Result_Data_64_bytes[11] := HwInputs.ST50_1_DM260_WPC_Result_Data_64_bytes[11];
	PlcInputs.ST50_1_DM260_WPC_Result_Data_64_bytes[12] := HwInputs.ST50_1_DM260_WPC_Result_Data_64_bytes[12];
	PlcInputs.ST50_1_DM260_WPC_Result_Data_64_bytes[13] := HwInputs.ST50_1_DM260_WPC_Result_Data_64_bytes[13];
	PlcInputs.ST50_1_DM260_WPC_Result_Data_64_bytes[14] := HwInputs.ST50_1_DM260_WPC_Result_Data_64_bytes[14];
	PlcInputs.ST50_1_DM260_WPC_Result_Data_64_bytes[15] := HwInputs.ST50_1_DM260_WPC_Result_Data_64_bytes[15];
	PlcInputs.ST50_1_DM260_WPC_Result_Data_64_bytes[16] := HwInputs.ST50_1_DM260_WPC_Result_Data_64_bytes[16];
	PlcInputs.ST50_1_DM260_WPC_Result_Data_64_bytes[17] := HwInputs.ST50_1_DM260_WPC_Result_Data_64_bytes[17];
	PlcInputs.ST50_1_DM260_WPC_Result_Data_64_bytes[18] := HwInputs.ST50_1_DM260_WPC_Result_Data_64_bytes[18];
	PlcInputs.ST50_1_DM260_WPC_Result_Data_64_bytes[19] := HwInputs.ST50_1_DM260_WPC_Result_Data_64_bytes[19];
	PlcInputs.ST50_1_DM260_WPC_Result_Data_64_bytes[20] := HwInputs.ST50_1_DM260_WPC_Result_Data_64_bytes[20];
	PlcInputs.ST50_1_DM260_WPC_Result_Data_64_bytes[21] := HwInputs.ST50_1_DM260_WPC_Result_Data_64_bytes[21];
	PlcInputs.ST50_1_DM260_WPC_Result_Data_64_bytes[22] := HwInputs.ST50_1_DM260_WPC_Result_Data_64_bytes[22];
	PlcInputs.ST50_1_DM260_WPC_Result_Data_64_bytes[23] := HwInputs.ST50_1_DM260_WPC_Result_Data_64_bytes[23];
	PlcInputs.ST50_1_DM260_WPC_Result_Data_64_bytes[24] := HwInputs.ST50_1_DM260_WPC_Result_Data_64_bytes[24];
	PlcInputs.ST50_1_DM260_WPC_Result_Data_64_bytes[25] := HwInputs.ST50_1_DM260_WPC_Result_Data_64_bytes[25];
	PlcInputs.ST50_1_DM260_WPC_Result_Data_64_bytes[26] := HwInputs.ST50_1_DM260_WPC_Result_Data_64_bytes[26];
	PlcInputs.ST50_1_DM260_WPC_Result_Data_64_bytes[27] := HwInputs.ST50_1_DM260_WPC_Result_Data_64_bytes[27];
	PlcInputs.ST50_1_DM260_WPC_Result_Data_64_bytes[28] := HwInputs.ST50_1_DM260_WPC_Result_Data_64_bytes[28];
	PlcInputs.ST50_1_DM260_WPC_Result_Data_64_bytes[29] := HwInputs.ST50_1_DM260_WPC_Result_Data_64_bytes[29];
	PlcInputs.ST50_1_DM260_WPC_Result_Data_64_bytes[30] := HwInputs.ST50_1_DM260_WPC_Result_Data_64_bytes[30];
	PlcInputs.ST50_1_DM260_WPC_Result_Data_64_bytes[31] := HwInputs.ST50_1_DM260_WPC_Result_Data_64_bytes[31];
	PlcInputs.ST50_1_DM260_WPC_Result_Data_64_bytes[32] := HwInputs.ST50_1_DM260_WPC_Result_Data_64_bytes[32];
	PlcInputs.ST50_1_DM260_WPC_Result_Data_64_bytes[33] := HwInputs.ST50_1_DM260_WPC_Result_Data_64_bytes[33];
	PlcInputs.ST50_1_DM260_WPC_Result_Data_64_bytes[34] := HwInputs.ST50_1_DM260_WPC_Result_Data_64_bytes[34];
	PlcInputs.ST50_1_DM260_WPC_Result_Data_64_bytes[35] := HwInputs.ST50_1_DM260_WPC_Result_Data_64_bytes[35];
	PlcInputs.ST50_1_DM260_WPC_Result_Data_64_bytes[36] := HwInputs.ST50_1_DM260_WPC_Result_Data_64_bytes[36];
	PlcInputs.ST50_1_DM260_WPC_Result_Data_64_bytes[37] := HwInputs.ST50_1_DM260_WPC_Result_Data_64_bytes[37];
	PlcInputs.ST50_1_DM260_WPC_Result_Data_64_bytes[38] := HwInputs.ST50_1_DM260_WPC_Result_Data_64_bytes[38];
	PlcInputs.ST50_1_DM260_WPC_Result_Data_64_bytes[39] := HwInputs.ST50_1_DM260_WPC_Result_Data_64_bytes[39];
	PlcInputs.ST50_1_DM260_WPC_Result_Data_64_bytes[40] := HwInputs.ST50_1_DM260_WPC_Result_Data_64_bytes[40];
	PlcInputs.ST50_1_DM260_WPC_Result_Data_64_bytes[41] := HwInputs.ST50_1_DM260_WPC_Result_Data_64_bytes[41];
	PlcInputs.ST50_1_DM260_WPC_Result_Data_64_bytes[42] := HwInputs.ST50_1_DM260_WPC_Result_Data_64_bytes[42];
	PlcInputs.ST50_1_DM260_WPC_Result_Data_64_bytes[43] := HwInputs.ST50_1_DM260_WPC_Result_Data_64_bytes[43];
	PlcInputs.ST50_1_DM260_WPC_Result_Data_64_bytes[44] := HwInputs.ST50_1_DM260_WPC_Result_Data_64_bytes[44];
	PlcInputs.ST50_1_DM260_WPC_Result_Data_64_bytes[45] := HwInputs.ST50_1_DM260_WPC_Result_Data_64_bytes[45];
	PlcInputs.ST50_1_DM260_WPC_Result_Data_64_bytes[46] := HwInputs.ST50_1_DM260_WPC_Result_Data_64_bytes[46];
	PlcInputs.ST50_1_DM260_WPC_Result_Data_64_bytes[47] := HwInputs.ST50_1_DM260_WPC_Result_Data_64_bytes[47];
	PlcInputs.ST50_1_DM260_WPC_Result_Data_64_bytes[48] := HwInputs.ST50_1_DM260_WPC_Result_Data_64_bytes[48];
	PlcInputs.ST50_1_DM260_WPC_Result_Data_64_bytes[49] := HwInputs.ST50_1_DM260_WPC_Result_Data_64_bytes[49];
	PlcInputs.ST50_1_DM260_WPC_Result_Data_64_bytes[50] := HwInputs.ST50_1_DM260_WPC_Result_Data_64_bytes[50];
	PlcInputs.ST50_1_DM260_WPC_Result_Data_64_bytes[51] := HwInputs.ST50_1_DM260_WPC_Result_Data_64_bytes[51];
	PlcInputs.ST50_1_DM260_WPC_Result_Data_64_bytes[52] := HwInputs.ST50_1_DM260_WPC_Result_Data_64_bytes[52];
	PlcInputs.ST50_1_DM260_WPC_Result_Data_64_bytes[53] := HwInputs.ST50_1_DM260_WPC_Result_Data_64_bytes[53];
	PlcInputs.ST50_1_DM260_WPC_Result_Data_64_bytes[54] := HwInputs.ST50_1_DM260_WPC_Result_Data_64_bytes[54];
	PlcInputs.ST50_1_DM260_WPC_Result_Data_64_bytes[55] := HwInputs.ST50_1_DM260_WPC_Result_Data_64_bytes[55];
	PlcInputs.ST50_1_DM260_WPC_Result_Data_64_bytes[56] := HwInputs.ST50_1_DM260_WPC_Result_Data_64_bytes[56];
	PlcInputs.ST50_1_DM260_WPC_Result_Data_64_bytes[57] := HwInputs.ST50_1_DM260_WPC_Result_Data_64_bytes[57];
	PlcInputs.ST50_1_DM260_WPC_Result_Data_64_bytes[58] := HwInputs.ST50_1_DM260_WPC_Result_Data_64_bytes[58];
	PlcInputs.ST50_1_DM260_WPC_Result_Data_64_bytes[59] := HwInputs.ST50_1_DM260_WPC_Result_Data_64_bytes[59];
	PlcInputs.ST50_1_DM260_WPC_Result_Data_64_bytes[60] := HwInputs.ST50_1_DM260_WPC_Result_Data_64_bytes[60];
	PlcInputs.ST50_1_DM260_WPC_Result_Data_64_bytes[61] := HwInputs.ST50_1_DM260_WPC_Result_Data_64_bytes[61];
	PlcInputs.ST50_1_DM260_WPC_Result_Data_64_bytes[62] := HwInputs.ST50_1_DM260_WPC_Result_Data_64_bytes[62];
	PlcInputs.ST50_1_DM260_WPC_Result_Data_64_bytes[63] := HwInputs.ST50_1_DM260_WPC_Result_Data_64_bytes[63];
	PlcInputs.ST50_1_DM260_WPC_Result_Data_64_bytes[64] := HwInputs.ST50_1_DM260_WPC_Result_Data_64_bytes[64];
	PlcInputs.ST50_1_DM260_WPC_Result_Data_64_bytes[65] := HwInputs.ST50_1_DM260_WPC_Result_Data_64_bytes[65];
	PlcInputs.ST50_1_DM260_WPC_Result_Data_64_bytes[66] := HwInputs.ST50_1_DM260_WPC_Result_Data_64_bytes[66];
	PlcInputs.ST50_1_DM260_WPC_Result_Data_64_bytes[67] := HwInputs.ST50_1_DM260_WPC_Result_Data_64_bytes[67];
	PlcInputs.ST50_1_DM260_WPC_Result_Data_64_bytes[68] := HwInputs.ST50_1_DM260_WPC_Result_Data_64_bytes[68];
	PlcInputs.ST50_1_DM260_WPC_Result_Data_64_bytes[69] := HwInputs.ST50_1_DM260_WPC_Result_Data_64_bytes[69];
	PlcInputs.ST50_1_DM260_WPC_Result_Data_64_bytes[70] := HwInputs.ST50_1_DM260_WPC_Result_Data_64_bytes[70];
	PlcInputs.ST50_1_DM260_WPC_Result_Data_64_bytes[71] := HwInputs.ST50_1_DM260_WPC_Result_Data_64_bytes[71];
	PlcInputs.ST50_1_DM260_Acquisition_Status[0] := HwInputs.ST50_1_DM260_Acquisition_Status[0];
	PlcInputs.ST50_1_DM260_Acquisition_Status[1] := HwInputs.ST50_1_DM260_Acquisition_Status[1];
	PlcInputs.ST50_1_DM260_Acquisition_Status[2] := HwInputs.ST50_1_DM260_Acquisition_Status[2];
	PlcInputs.ST50_1_DM260_Results_Status := HwInputs.ST50_1_DM260_Results_Status;
	PlcInputs.ST50_1_DM260_Soft_Event_Control := HwInputs.ST50_1_DM260_Soft_Event_Control;
	PlcInputs.ST50_1_DM260_Result_Data_64_bytes[0] := HwInputs.ST50_1_DM260_Result_Data_64_bytes[0];
	PlcInputs.ST50_1_DM260_Result_Data_64_bytes[1] := HwInputs.ST50_1_DM260_Result_Data_64_bytes[1];
	PlcInputs.ST50_1_DM260_Result_Data_64_bytes[2] := HwInputs.ST50_1_DM260_Result_Data_64_bytes[2];
	PlcInputs.ST50_1_DM260_Result_Data_64_bytes[3] := HwInputs.ST50_1_DM260_Result_Data_64_bytes[3];
	PlcInputs.ST50_1_DM260_Result_Data_64_bytes[4] := HwInputs.ST50_1_DM260_Result_Data_64_bytes[4];
	PlcInputs.ST50_1_DM260_Result_Data_64_bytes[5] := HwInputs.ST50_1_DM260_Result_Data_64_bytes[5];
	PlcInputs.ST50_1_DM260_Result_Data_64_bytes[6] := HwInputs.ST50_1_DM260_Result_Data_64_bytes[6];
	PlcInputs.ST50_1_DM260_Result_Data_64_bytes[7] := HwInputs.ST50_1_DM260_Result_Data_64_bytes[7];
	PlcInputs.ST50_1_DM260_Result_Data_64_bytes[8] := HwInputs.ST50_1_DM260_Result_Data_64_bytes[8];
	PlcInputs.ST50_1_DM260_Result_Data_64_bytes[9] := HwInputs.ST50_1_DM260_Result_Data_64_bytes[9];
	PlcInputs.ST50_1_DM260_Result_Data_64_bytes[10] := HwInputs.ST50_1_DM260_Result_Data_64_bytes[10];
	PlcInputs.ST50_1_DM260_Result_Data_64_bytes[11] := HwInputs.ST50_1_DM260_Result_Data_64_bytes[11];
	PlcInputs.ST50_1_DM260_Result_Data_64_bytes[12] := HwInputs.ST50_1_DM260_Result_Data_64_bytes[12];
	PlcInputs.ST50_1_DM260_Result_Data_64_bytes[13] := HwInputs.ST50_1_DM260_Result_Data_64_bytes[13];
	PlcInputs.ST50_1_DM260_Result_Data_64_bytes[14] := HwInputs.ST50_1_DM260_Result_Data_64_bytes[14];
	PlcInputs.ST50_1_DM260_Result_Data_64_bytes[15] := HwInputs.ST50_1_DM260_Result_Data_64_bytes[15];
	PlcInputs.ST50_1_DM260_Result_Data_64_bytes[16] := HwInputs.ST50_1_DM260_Result_Data_64_bytes[16];
	PlcInputs.ST50_1_DM260_Result_Data_64_bytes[17] := HwInputs.ST50_1_DM260_Result_Data_64_bytes[17];
	PlcInputs.ST50_1_DM260_Result_Data_64_bytes[18] := HwInputs.ST50_1_DM260_Result_Data_64_bytes[18];
	PlcInputs.ST50_1_DM260_Result_Data_64_bytes[19] := HwInputs.ST50_1_DM260_Result_Data_64_bytes[19];
	PlcInputs.ST50_1_DM260_Result_Data_64_bytes[20] := HwInputs.ST50_1_DM260_Result_Data_64_bytes[20];
	PlcInputs.ST50_1_DM260_Result_Data_64_bytes[21] := HwInputs.ST50_1_DM260_Result_Data_64_bytes[21];
	PlcInputs.ST50_1_DM260_Result_Data_64_bytes[22] := HwInputs.ST50_1_DM260_Result_Data_64_bytes[22];
	PlcInputs.ST50_1_DM260_Result_Data_64_bytes[23] := HwInputs.ST50_1_DM260_Result_Data_64_bytes[23];
	PlcInputs.ST50_1_DM260_Result_Data_64_bytes[24] := HwInputs.ST50_1_DM260_Result_Data_64_bytes[24];
	PlcInputs.ST50_1_DM260_Result_Data_64_bytes[25] := HwInputs.ST50_1_DM260_Result_Data_64_bytes[25];
	PlcInputs.ST50_1_DM260_Result_Data_64_bytes[26] := HwInputs.ST50_1_DM260_Result_Data_64_bytes[26];
	PlcInputs.ST50_1_DM260_Result_Data_64_bytes[27] := HwInputs.ST50_1_DM260_Result_Data_64_bytes[27];
	PlcInputs.ST50_1_DM260_Result_Data_64_bytes[28] := HwInputs.ST50_1_DM260_Result_Data_64_bytes[28];
	PlcInputs.ST50_1_DM260_Result_Data_64_bytes[29] := HwInputs.ST50_1_DM260_Result_Data_64_bytes[29];
	PlcInputs.ST50_1_DM260_Result_Data_64_bytes[30] := HwInputs.ST50_1_DM260_Result_Data_64_bytes[30];
	PlcInputs.ST50_1_DM260_Result_Data_64_bytes[31] := HwInputs.ST50_1_DM260_Result_Data_64_bytes[31];
	PlcInputs.ST50_1_DM260_Result_Data_64_bytes[32] := HwInputs.ST50_1_DM260_Result_Data_64_bytes[32];
	PlcInputs.ST50_1_DM260_Result_Data_64_bytes[33] := HwInputs.ST50_1_DM260_Result_Data_64_bytes[33];
	PlcInputs.ST50_1_DM260_Result_Data_64_bytes[34] := HwInputs.ST50_1_DM260_Result_Data_64_bytes[34];
	PlcInputs.ST50_1_DM260_Result_Data_64_bytes[35] := HwInputs.ST50_1_DM260_Result_Data_64_bytes[35];
	PlcInputs.ST50_1_DM260_Result_Data_64_bytes[36] := HwInputs.ST50_1_DM260_Result_Data_64_bytes[36];
	PlcInputs.ST50_1_DM260_Result_Data_64_bytes[37] := HwInputs.ST50_1_DM260_Result_Data_64_bytes[37];
	PlcInputs.ST50_1_DM260_Result_Data_64_bytes[38] := HwInputs.ST50_1_DM260_Result_Data_64_bytes[38];
	PlcInputs.ST50_1_DM260_Result_Data_64_bytes[39] := HwInputs.ST50_1_DM260_Result_Data_64_bytes[39];
	PlcInputs.ST50_1_DM260_Result_Data_64_bytes[40] := HwInputs.ST50_1_DM260_Result_Data_64_bytes[40];
	PlcInputs.ST50_1_DM260_Result_Data_64_bytes[41] := HwInputs.ST50_1_DM260_Result_Data_64_bytes[41];
	PlcInputs.ST50_1_DM260_Result_Data_64_bytes[42] := HwInputs.ST50_1_DM260_Result_Data_64_bytes[42];
	PlcInputs.ST50_1_DM260_Result_Data_64_bytes[43] := HwInputs.ST50_1_DM260_Result_Data_64_bytes[43];
	PlcInputs.ST50_1_DM260_Result_Data_64_bytes[44] := HwInputs.ST50_1_DM260_Result_Data_64_bytes[44];
	PlcInputs.ST50_1_DM260_Result_Data_64_bytes[45] := HwInputs.ST50_1_DM260_Result_Data_64_bytes[45];
	PlcInputs.ST50_1_DM260_Result_Data_64_bytes[46] := HwInputs.ST50_1_DM260_Result_Data_64_bytes[46];
	PlcInputs.ST50_1_DM260_Result_Data_64_bytes[47] := HwInputs.ST50_1_DM260_Result_Data_64_bytes[47];
	PlcInputs.ST50_1_DM260_Result_Data_64_bytes[48] := HwInputs.ST50_1_DM260_Result_Data_64_bytes[48];
	PlcInputs.ST50_1_DM260_Result_Data_64_bytes[49] := HwInputs.ST50_1_DM260_Result_Data_64_bytes[49];
	PlcInputs.ST50_1_DM260_Result_Data_64_bytes[50] := HwInputs.ST50_1_DM260_Result_Data_64_bytes[50];
	PlcInputs.ST50_1_DM260_Result_Data_64_bytes[51] := HwInputs.ST50_1_DM260_Result_Data_64_bytes[51];
	PlcInputs.ST50_1_DM260_Result_Data_64_bytes[52] := HwInputs.ST50_1_DM260_Result_Data_64_bytes[52];
	PlcInputs.ST50_1_DM260_Result_Data_64_bytes[53] := HwInputs.ST50_1_DM260_Result_Data_64_bytes[53];
	PlcInputs.ST50_1_DM260_Result_Data_64_bytes[54] := HwInputs.ST50_1_DM260_Result_Data_64_bytes[54];
	PlcInputs.ST50_1_DM260_Result_Data_64_bytes[55] := HwInputs.ST50_1_DM260_Result_Data_64_bytes[55];
	PlcInputs.ST50_1_DM260_Result_Data_64_bytes[56] := HwInputs.ST50_1_DM260_Result_Data_64_bytes[56];
	PlcInputs.ST50_1_DM260_Result_Data_64_bytes[57] := HwInputs.ST50_1_DM260_Result_Data_64_bytes[57];
	PlcInputs.ST50_1_DM260_Result_Data_64_bytes[58] := HwInputs.ST50_1_DM260_Result_Data_64_bytes[58];
	PlcInputs.ST50_1_DM260_Result_Data_64_bytes[59] := HwInputs.ST50_1_DM260_Result_Data_64_bytes[59];
	PlcInputs.ST50_1_DM260_Result_Data_64_bytes[60] := HwInputs.ST50_1_DM260_Result_Data_64_bytes[60];
	PlcInputs.ST50_1_DM260_Result_Data_64_bytes[61] := HwInputs.ST50_1_DM260_Result_Data_64_bytes[61];
	PlcInputs.ST50_1_DM260_Result_Data_64_bytes[62] := HwInputs.ST50_1_DM260_Result_Data_64_bytes[62];
	PlcInputs.ST50_1_DM260_Result_Data_64_bytes[63] := HwInputs.ST50_1_DM260_Result_Data_64_bytes[63];
	PlcInputs.ST50_1_DM260_Result_Data_64_bytes[64] := HwInputs.ST50_1_DM260_Result_Data_64_bytes[64];
	PlcInputs.ST50_1_DM260_Result_Data_64_bytes[65] := HwInputs.ST50_1_DM260_Result_Data_64_bytes[65];
	PlcInputs.ST50_1_DM260_Result_Data_64_bytes[66] := HwInputs.ST50_1_DM260_Result_Data_64_bytes[66];
	PlcInputs.ST50_1_DM260_Result_Data_64_bytes[67] := HwInputs.ST50_1_DM260_Result_Data_64_bytes[67];
	PlcInputs.ST50_1_DM260_Result_Data_64_bytes[68] := HwInputs.ST50_1_DM260_Result_Data_64_bytes[68];
	PlcInputs.ST50_1_DM260_Result_Data_64_bytes[69] := HwInputs.ST50_1_DM260_Result_Data_64_bytes[69];
	PlcInputs.ST50_1_DM260_Result_Data_64_bytes[70] := HwInputs.ST50_1_DM260_Result_Data_64_bytes[70];
	PlcInputs.ST50_1_DM260_Result_Data_64_bytes[71] := HwInputs.ST50_1_DM260_Result_Data_64_bytes[71];
	PlcInputs.ST50_2_DM260_Acquisition_Status[0] := HwInputs.ST50_2_DM260_Acquisition_Status[0];
	PlcInputs.ST50_2_DM260_Acquisition_Status[1] := HwInputs.ST50_2_DM260_Acquisition_Status[1];
	PlcInputs.ST50_2_DM260_Acquisition_Status[2] := HwInputs.ST50_2_DM260_Acquisition_Status[2];
	PlcInputs.ST50_2_DM260_Results_Status := HwInputs.ST50_2_DM260_Results_Status;
	PlcInputs.ST50_2_DM260_Soft_Event_Control := HwInputs.ST50_2_DM260_Soft_Event_Control;
	PlcInputs.ST50_2_DM260_Result_Data_64_bytes[0] := HwInputs.ST50_2_DM260_Result_Data_64_bytes[0];
	PlcInputs.ST50_2_DM260_Result_Data_64_bytes[1] := HwInputs.ST50_2_DM260_Result_Data_64_bytes[1];
	PlcInputs.ST50_2_DM260_Result_Data_64_bytes[2] := HwInputs.ST50_2_DM260_Result_Data_64_bytes[2];
	PlcInputs.ST50_2_DM260_Result_Data_64_bytes[3] := HwInputs.ST50_2_DM260_Result_Data_64_bytes[3];
	PlcInputs.ST50_2_DM260_Result_Data_64_bytes[4] := HwInputs.ST50_2_DM260_Result_Data_64_bytes[4];
	PlcInputs.ST50_2_DM260_Result_Data_64_bytes[5] := HwInputs.ST50_2_DM260_Result_Data_64_bytes[5];
	PlcInputs.ST50_2_DM260_Result_Data_64_bytes[6] := HwInputs.ST50_2_DM260_Result_Data_64_bytes[6];
	PlcInputs.ST50_2_DM260_Result_Data_64_bytes[7] := HwInputs.ST50_2_DM260_Result_Data_64_bytes[7];
	PlcInputs.ST50_2_DM260_Result_Data_64_bytes[8] := HwInputs.ST50_2_DM260_Result_Data_64_bytes[8];
	PlcInputs.ST50_2_DM260_Result_Data_64_bytes[9] := HwInputs.ST50_2_DM260_Result_Data_64_bytes[9];
	PlcInputs.ST50_2_DM260_Result_Data_64_bytes[10] := HwInputs.ST50_2_DM260_Result_Data_64_bytes[10];
	PlcInputs.ST50_2_DM260_Result_Data_64_bytes[11] := HwInputs.ST50_2_DM260_Result_Data_64_bytes[11];
	PlcInputs.ST50_2_DM260_Result_Data_64_bytes[12] := HwInputs.ST50_2_DM260_Result_Data_64_bytes[12];
	PlcInputs.ST50_2_DM260_Result_Data_64_bytes[13] := HwInputs.ST50_2_DM260_Result_Data_64_bytes[13];
	PlcInputs.ST50_2_DM260_Result_Data_64_bytes[14] := HwInputs.ST50_2_DM260_Result_Data_64_bytes[14];
	PlcInputs.ST50_2_DM260_Result_Data_64_bytes[15] := HwInputs.ST50_2_DM260_Result_Data_64_bytes[15];
	PlcInputs.ST50_2_DM260_Result_Data_64_bytes[16] := HwInputs.ST50_2_DM260_Result_Data_64_bytes[16];
	PlcInputs.ST50_2_DM260_Result_Data_64_bytes[17] := HwInputs.ST50_2_DM260_Result_Data_64_bytes[17];
	PlcInputs.ST50_2_DM260_Result_Data_64_bytes[18] := HwInputs.ST50_2_DM260_Result_Data_64_bytes[18];
	PlcInputs.ST50_2_DM260_Result_Data_64_bytes[19] := HwInputs.ST50_2_DM260_Result_Data_64_bytes[19];
	PlcInputs.ST50_2_DM260_Result_Data_64_bytes[20] := HwInputs.ST50_2_DM260_Result_Data_64_bytes[20];
	PlcInputs.ST50_2_DM260_Result_Data_64_bytes[21] := HwInputs.ST50_2_DM260_Result_Data_64_bytes[21];
	PlcInputs.ST50_2_DM260_Result_Data_64_bytes[22] := HwInputs.ST50_2_DM260_Result_Data_64_bytes[22];
	PlcInputs.ST50_2_DM260_Result_Data_64_bytes[23] := HwInputs.ST50_2_DM260_Result_Data_64_bytes[23];
	PlcInputs.ST50_2_DM260_Result_Data_64_bytes[24] := HwInputs.ST50_2_DM260_Result_Data_64_bytes[24];
	PlcInputs.ST50_2_DM260_Result_Data_64_bytes[25] := HwInputs.ST50_2_DM260_Result_Data_64_bytes[25];
	PlcInputs.ST50_2_DM260_Result_Data_64_bytes[26] := HwInputs.ST50_2_DM260_Result_Data_64_bytes[26];
	PlcInputs.ST50_2_DM260_Result_Data_64_bytes[27] := HwInputs.ST50_2_DM260_Result_Data_64_bytes[27];
	PlcInputs.ST50_2_DM260_Result_Data_64_bytes[28] := HwInputs.ST50_2_DM260_Result_Data_64_bytes[28];
	PlcInputs.ST50_2_DM260_Result_Data_64_bytes[29] := HwInputs.ST50_2_DM260_Result_Data_64_bytes[29];
	PlcInputs.ST50_2_DM260_Result_Data_64_bytes[30] := HwInputs.ST50_2_DM260_Result_Data_64_bytes[30];
	PlcInputs.ST50_2_DM260_Result_Data_64_bytes[31] := HwInputs.ST50_2_DM260_Result_Data_64_bytes[31];
	PlcInputs.ST50_2_DM260_Result_Data_64_bytes[32] := HwInputs.ST50_2_DM260_Result_Data_64_bytes[32];
	PlcInputs.ST50_2_DM260_Result_Data_64_bytes[33] := HwInputs.ST50_2_DM260_Result_Data_64_bytes[33];
	PlcInputs.ST50_2_DM260_Result_Data_64_bytes[34] := HwInputs.ST50_2_DM260_Result_Data_64_bytes[34];
	PlcInputs.ST50_2_DM260_Result_Data_64_bytes[35] := HwInputs.ST50_2_DM260_Result_Data_64_bytes[35];
	PlcInputs.ST50_2_DM260_Result_Data_64_bytes[36] := HwInputs.ST50_2_DM260_Result_Data_64_bytes[36];
	PlcInputs.ST50_2_DM260_Result_Data_64_bytes[37] := HwInputs.ST50_2_DM260_Result_Data_64_bytes[37];
	PlcInputs.ST50_2_DM260_Result_Data_64_bytes[38] := HwInputs.ST50_2_DM260_Result_Data_64_bytes[38];
	PlcInputs.ST50_2_DM260_Result_Data_64_bytes[39] := HwInputs.ST50_2_DM260_Result_Data_64_bytes[39];
	PlcInputs.ST50_2_DM260_Result_Data_64_bytes[40] := HwInputs.ST50_2_DM260_Result_Data_64_bytes[40];
	PlcInputs.ST50_2_DM260_Result_Data_64_bytes[41] := HwInputs.ST50_2_DM260_Result_Data_64_bytes[41];
	PlcInputs.ST50_2_DM260_Result_Data_64_bytes[42] := HwInputs.ST50_2_DM260_Result_Data_64_bytes[42];
	PlcInputs.ST50_2_DM260_Result_Data_64_bytes[43] := HwInputs.ST50_2_DM260_Result_Data_64_bytes[43];
	PlcInputs.ST50_2_DM260_Result_Data_64_bytes[44] := HwInputs.ST50_2_DM260_Result_Data_64_bytes[44];
	PlcInputs.ST50_2_DM260_Result_Data_64_bytes[45] := HwInputs.ST50_2_DM260_Result_Data_64_bytes[45];
	PlcInputs.ST50_2_DM260_Result_Data_64_bytes[46] := HwInputs.ST50_2_DM260_Result_Data_64_bytes[46];
	PlcInputs.ST50_2_DM260_Result_Data_64_bytes[47] := HwInputs.ST50_2_DM260_Result_Data_64_bytes[47];
	PlcInputs.ST50_2_DM260_Result_Data_64_bytes[48] := HwInputs.ST50_2_DM260_Result_Data_64_bytes[48];
	PlcInputs.ST50_2_DM260_Result_Data_64_bytes[49] := HwInputs.ST50_2_DM260_Result_Data_64_bytes[49];
	PlcInputs.ST50_2_DM260_Result_Data_64_bytes[50] := HwInputs.ST50_2_DM260_Result_Data_64_bytes[50];
	PlcInputs.ST50_2_DM260_Result_Data_64_bytes[51] := HwInputs.ST50_2_DM260_Result_Data_64_bytes[51];
	PlcInputs.ST50_2_DM260_Result_Data_64_bytes[52] := HwInputs.ST50_2_DM260_Result_Data_64_bytes[52];
	PlcInputs.ST50_2_DM260_Result_Data_64_bytes[53] := HwInputs.ST50_2_DM260_Result_Data_64_bytes[53];
	PlcInputs.ST50_2_DM260_Result_Data_64_bytes[54] := HwInputs.ST50_2_DM260_Result_Data_64_bytes[54];
	PlcInputs.ST50_2_DM260_Result_Data_64_bytes[55] := HwInputs.ST50_2_DM260_Result_Data_64_bytes[55];
	PlcInputs.ST50_2_DM260_Result_Data_64_bytes[56] := HwInputs.ST50_2_DM260_Result_Data_64_bytes[56];
	PlcInputs.ST50_2_DM260_Result_Data_64_bytes[57] := HwInputs.ST50_2_DM260_Result_Data_64_bytes[57];
	PlcInputs.ST50_2_DM260_Result_Data_64_bytes[58] := HwInputs.ST50_2_DM260_Result_Data_64_bytes[58];
	PlcInputs.ST50_2_DM260_Result_Data_64_bytes[59] := HwInputs.ST50_2_DM260_Result_Data_64_bytes[59];
	PlcInputs.ST50_2_DM260_Result_Data_64_bytes[60] := HwInputs.ST50_2_DM260_Result_Data_64_bytes[60];
	PlcInputs.ST50_2_DM260_Result_Data_64_bytes[61] := HwInputs.ST50_2_DM260_Result_Data_64_bytes[61];
	PlcInputs.ST50_2_DM260_Result_Data_64_bytes[62] := HwInputs.ST50_2_DM260_Result_Data_64_bytes[62];
	PlcInputs.ST50_2_DM260_Result_Data_64_bytes[63] := HwInputs.ST50_2_DM260_Result_Data_64_bytes[63];
	PlcInputs.ST50_2_DM260_Result_Data_64_bytes[64] := HwInputs.ST50_2_DM260_Result_Data_64_bytes[64];
	PlcInputs.ST50_2_DM260_Result_Data_64_bytes[65] := HwInputs.ST50_2_DM260_Result_Data_64_bytes[65];
	PlcInputs.ST50_2_DM260_Result_Data_64_bytes[66] := HwInputs.ST50_2_DM260_Result_Data_64_bytes[66];
	PlcInputs.ST50_2_DM260_Result_Data_64_bytes[67] := HwInputs.ST50_2_DM260_Result_Data_64_bytes[67];
	PlcInputs.ST50_2_DM260_Result_Data_64_bytes[68] := HwInputs.ST50_2_DM260_Result_Data_64_bytes[68];
	PlcInputs.ST50_2_DM260_Result_Data_64_bytes[69] := HwInputs.ST50_2_DM260_Result_Data_64_bytes[69];
	PlcInputs.ST50_2_DM260_Result_Data_64_bytes[70] := HwInputs.ST50_2_DM260_Result_Data_64_bytes[70];
	PlcInputs.ST50_2_DM260_Result_Data_64_bytes[71] := HwInputs.ST50_2_DM260_Result_Data_64_bytes[71];
	PlcInputs.ST50_3_DM260_Acquisition_Status[0] := HwInputs.ST50_3_DM260_Acquisition_Status[0];
	PlcInputs.ST50_3_DM260_Acquisition_Status[1] := HwInputs.ST50_3_DM260_Acquisition_Status[1];
	PlcInputs.ST50_3_DM260_Acquisition_Status[2] := HwInputs.ST50_3_DM260_Acquisition_Status[2];
	PlcInputs.ST50_3_DM260_Results_Status := HwInputs.ST50_3_DM260_Results_Status;
	PlcInputs.ST50_3_DM260_Soft_Event_Control := HwInputs.ST50_3_DM260_Soft_Event_Control;
	PlcInputs.ST50_3_DM260_Result_Data_64_bytes[0] := HwInputs.ST50_3_DM260_Result_Data_64_bytes[0];
	PlcInputs.ST50_3_DM260_Result_Data_64_bytes[1] := HwInputs.ST50_3_DM260_Result_Data_64_bytes[1];
	PlcInputs.ST50_3_DM260_Result_Data_64_bytes[2] := HwInputs.ST50_3_DM260_Result_Data_64_bytes[2];
	PlcInputs.ST50_3_DM260_Result_Data_64_bytes[3] := HwInputs.ST50_3_DM260_Result_Data_64_bytes[3];
	PlcInputs.ST50_3_DM260_Result_Data_64_bytes[4] := HwInputs.ST50_3_DM260_Result_Data_64_bytes[4];
	PlcInputs.ST50_3_DM260_Result_Data_64_bytes[5] := HwInputs.ST50_3_DM260_Result_Data_64_bytes[5];
	PlcInputs.ST50_3_DM260_Result_Data_64_bytes[6] := HwInputs.ST50_3_DM260_Result_Data_64_bytes[6];
	PlcInputs.ST50_3_DM260_Result_Data_64_bytes[7] := HwInputs.ST50_3_DM260_Result_Data_64_bytes[7];
	PlcInputs.ST50_3_DM260_Result_Data_64_bytes[8] := HwInputs.ST50_3_DM260_Result_Data_64_bytes[8];
	PlcInputs.ST50_3_DM260_Result_Data_64_bytes[9] := HwInputs.ST50_3_DM260_Result_Data_64_bytes[9];
	PlcInputs.ST50_3_DM260_Result_Data_64_bytes[10] := HwInputs.ST50_3_DM260_Result_Data_64_bytes[10];
	PlcInputs.ST50_3_DM260_Result_Data_64_bytes[11] := HwInputs.ST50_3_DM260_Result_Data_64_bytes[11];
	PlcInputs.ST50_3_DM260_Result_Data_64_bytes[12] := HwInputs.ST50_3_DM260_Result_Data_64_bytes[12];
	PlcInputs.ST50_3_DM260_Result_Data_64_bytes[13] := HwInputs.ST50_3_DM260_Result_Data_64_bytes[13];
	PlcInputs.ST50_3_DM260_Result_Data_64_bytes[14] := HwInputs.ST50_3_DM260_Result_Data_64_bytes[14];
	PlcInputs.ST50_3_DM260_Result_Data_64_bytes[15] := HwInputs.ST50_3_DM260_Result_Data_64_bytes[15];
	PlcInputs.ST50_3_DM260_Result_Data_64_bytes[16] := HwInputs.ST50_3_DM260_Result_Data_64_bytes[16];
	PlcInputs.ST50_3_DM260_Result_Data_64_bytes[17] := HwInputs.ST50_3_DM260_Result_Data_64_bytes[17];
	PlcInputs.ST50_3_DM260_Result_Data_64_bytes[18] := HwInputs.ST50_3_DM260_Result_Data_64_bytes[18];
	PlcInputs.ST50_3_DM260_Result_Data_64_bytes[19] := HwInputs.ST50_3_DM260_Result_Data_64_bytes[19];
	PlcInputs.ST50_3_DM260_Result_Data_64_bytes[20] := HwInputs.ST50_3_DM260_Result_Data_64_bytes[20];
	PlcInputs.ST50_3_DM260_Result_Data_64_bytes[21] := HwInputs.ST50_3_DM260_Result_Data_64_bytes[21];
	PlcInputs.ST50_3_DM260_Result_Data_64_bytes[22] := HwInputs.ST50_3_DM260_Result_Data_64_bytes[22];
	PlcInputs.ST50_3_DM260_Result_Data_64_bytes[23] := HwInputs.ST50_3_DM260_Result_Data_64_bytes[23];
	PlcInputs.ST50_3_DM260_Result_Data_64_bytes[24] := HwInputs.ST50_3_DM260_Result_Data_64_bytes[24];
	PlcInputs.ST50_3_DM260_Result_Data_64_bytes[25] := HwInputs.ST50_3_DM260_Result_Data_64_bytes[25];
	PlcInputs.ST50_3_DM260_Result_Data_64_bytes[26] := HwInputs.ST50_3_DM260_Result_Data_64_bytes[26];
	PlcInputs.ST50_3_DM260_Result_Data_64_bytes[27] := HwInputs.ST50_3_DM260_Result_Data_64_bytes[27];
	PlcInputs.ST50_3_DM260_Result_Data_64_bytes[28] := HwInputs.ST50_3_DM260_Result_Data_64_bytes[28];
	PlcInputs.ST50_3_DM260_Result_Data_64_bytes[29] := HwInputs.ST50_3_DM260_Result_Data_64_bytes[29];
	PlcInputs.ST50_3_DM260_Result_Data_64_bytes[30] := HwInputs.ST50_3_DM260_Result_Data_64_bytes[30];
	PlcInputs.ST50_3_DM260_Result_Data_64_bytes[31] := HwInputs.ST50_3_DM260_Result_Data_64_bytes[31];
	PlcInputs.ST50_3_DM260_Result_Data_64_bytes[32] := HwInputs.ST50_3_DM260_Result_Data_64_bytes[32];
	PlcInputs.ST50_3_DM260_Result_Data_64_bytes[33] := HwInputs.ST50_3_DM260_Result_Data_64_bytes[33];
	PlcInputs.ST50_3_DM260_Result_Data_64_bytes[34] := HwInputs.ST50_3_DM260_Result_Data_64_bytes[34];
	PlcInputs.ST50_3_DM260_Result_Data_64_bytes[35] := HwInputs.ST50_3_DM260_Result_Data_64_bytes[35];
	PlcInputs.ST50_3_DM260_Result_Data_64_bytes[36] := HwInputs.ST50_3_DM260_Result_Data_64_bytes[36];
	PlcInputs.ST50_3_DM260_Result_Data_64_bytes[37] := HwInputs.ST50_3_DM260_Result_Data_64_bytes[37];
	PlcInputs.ST50_3_DM260_Result_Data_64_bytes[38] := HwInputs.ST50_3_DM260_Result_Data_64_bytes[38];
	PlcInputs.ST50_3_DM260_Result_Data_64_bytes[39] := HwInputs.ST50_3_DM260_Result_Data_64_bytes[39];
	PlcInputs.ST50_3_DM260_Result_Data_64_bytes[40] := HwInputs.ST50_3_DM260_Result_Data_64_bytes[40];
	PlcInputs.ST50_3_DM260_Result_Data_64_bytes[41] := HwInputs.ST50_3_DM260_Result_Data_64_bytes[41];
	PlcInputs.ST50_3_DM260_Result_Data_64_bytes[42] := HwInputs.ST50_3_DM260_Result_Data_64_bytes[42];
	PlcInputs.ST50_3_DM260_Result_Data_64_bytes[43] := HwInputs.ST50_3_DM260_Result_Data_64_bytes[43];
	PlcInputs.ST50_3_DM260_Result_Data_64_bytes[44] := HwInputs.ST50_3_DM260_Result_Data_64_bytes[44];
	PlcInputs.ST50_3_DM260_Result_Data_64_bytes[45] := HwInputs.ST50_3_DM260_Result_Data_64_bytes[45];
	PlcInputs.ST50_3_DM260_Result_Data_64_bytes[46] := HwInputs.ST50_3_DM260_Result_Data_64_bytes[46];
	PlcInputs.ST50_3_DM260_Result_Data_64_bytes[47] := HwInputs.ST50_3_DM260_Result_Data_64_bytes[47];
	PlcInputs.ST50_3_DM260_Result_Data_64_bytes[48] := HwInputs.ST50_3_DM260_Result_Data_64_bytes[48];
	PlcInputs.ST50_3_DM260_Result_Data_64_bytes[49] := HwInputs.ST50_3_DM260_Result_Data_64_bytes[49];
	PlcInputs.ST50_3_DM260_Result_Data_64_bytes[50] := HwInputs.ST50_3_DM260_Result_Data_64_bytes[50];
	PlcInputs.ST50_3_DM260_Result_Data_64_bytes[51] := HwInputs.ST50_3_DM260_Result_Data_64_bytes[51];
	PlcInputs.ST50_3_DM260_Result_Data_64_bytes[52] := HwInputs.ST50_3_DM260_Result_Data_64_bytes[52];
	PlcInputs.ST50_3_DM260_Result_Data_64_bytes[53] := HwInputs.ST50_3_DM260_Result_Data_64_bytes[53];
	PlcInputs.ST50_3_DM260_Result_Data_64_bytes[54] := HwInputs.ST50_3_DM260_Result_Data_64_bytes[54];
	PlcInputs.ST50_3_DM260_Result_Data_64_bytes[55] := HwInputs.ST50_3_DM260_Result_Data_64_bytes[55];
	PlcInputs.ST50_3_DM260_Result_Data_64_bytes[56] := HwInputs.ST50_3_DM260_Result_Data_64_bytes[56];
	PlcInputs.ST50_3_DM260_Result_Data_64_bytes[57] := HwInputs.ST50_3_DM260_Result_Data_64_bytes[57];
	PlcInputs.ST50_3_DM260_Result_Data_64_bytes[58] := HwInputs.ST50_3_DM260_Result_Data_64_bytes[58];
	PlcInputs.ST50_3_DM260_Result_Data_64_bytes[59] := HwInputs.ST50_3_DM260_Result_Data_64_bytes[59];
	PlcInputs.ST50_3_DM260_Result_Data_64_bytes[60] := HwInputs.ST50_3_DM260_Result_Data_64_bytes[60];
	PlcInputs.ST50_3_DM260_Result_Data_64_bytes[61] := HwInputs.ST50_3_DM260_Result_Data_64_bytes[61];
	PlcInputs.ST50_3_DM260_Result_Data_64_bytes[62] := HwInputs.ST50_3_DM260_Result_Data_64_bytes[62];
	PlcInputs.ST50_3_DM260_Result_Data_64_bytes[63] := HwInputs.ST50_3_DM260_Result_Data_64_bytes[63];
	PlcInputs.ST50_3_DM260_Result_Data_64_bytes[64] := HwInputs.ST50_3_DM260_Result_Data_64_bytes[64];
	PlcInputs.ST50_3_DM260_Result_Data_64_bytes[65] := HwInputs.ST50_3_DM260_Result_Data_64_bytes[65];
	PlcInputs.ST50_3_DM260_Result_Data_64_bytes[66] := HwInputs.ST50_3_DM260_Result_Data_64_bytes[66];
	PlcInputs.ST50_3_DM260_Result_Data_64_bytes[67] := HwInputs.ST50_3_DM260_Result_Data_64_bytes[67];
	PlcInputs.ST50_3_DM260_Result_Data_64_bytes[68] := HwInputs.ST50_3_DM260_Result_Data_64_bytes[68];
	PlcInputs.ST50_3_DM260_Result_Data_64_bytes[69] := HwInputs.ST50_3_DM260_Result_Data_64_bytes[69];
	PlcInputs.ST50_3_DM260_Result_Data_64_bytes[70] := HwInputs.ST50_3_DM260_Result_Data_64_bytes[70];
	PlcInputs.ST50_3_DM260_Result_Data_64_bytes[71] := HwInputs.ST50_3_DM260_Result_Data_64_bytes[71];
	PlcInputs.ST50_4_DM260_Acquisition_Status[0] := HwInputs.ST50_4_DM260_Acquisition_Status[0];
	PlcInputs.ST50_4_DM260_Acquisition_Status[1] := HwInputs.ST50_4_DM260_Acquisition_Status[1];
	PlcInputs.ST50_4_DM260_Acquisition_Status[2] := HwInputs.ST50_4_DM260_Acquisition_Status[2];
	PlcInputs.ST50_4_DM260_Results_Status := HwInputs.ST50_4_DM260_Results_Status;
	PlcInputs.ST50_4_DM260_Soft_Event_Control := HwInputs.ST50_4_DM260_Soft_Event_Control;
	PlcInputs.ST50_4_DM260_Result_Data_64_bytes[0] := HwInputs.ST50_4_DM260_Result_Data_64_bytes[0];
	PlcInputs.ST50_4_DM260_Result_Data_64_bytes[1] := HwInputs.ST50_4_DM260_Result_Data_64_bytes[1];
	PlcInputs.ST50_4_DM260_Result_Data_64_bytes[2] := HwInputs.ST50_4_DM260_Result_Data_64_bytes[2];
	PlcInputs.ST50_4_DM260_Result_Data_64_bytes[3] := HwInputs.ST50_4_DM260_Result_Data_64_bytes[3];
	PlcInputs.ST50_4_DM260_Result_Data_64_bytes[4] := HwInputs.ST50_4_DM260_Result_Data_64_bytes[4];
	PlcInputs.ST50_4_DM260_Result_Data_64_bytes[5] := HwInputs.ST50_4_DM260_Result_Data_64_bytes[5];
	PlcInputs.ST50_4_DM260_Result_Data_64_bytes[6] := HwInputs.ST50_4_DM260_Result_Data_64_bytes[6];
	PlcInputs.ST50_4_DM260_Result_Data_64_bytes[7] := HwInputs.ST50_4_DM260_Result_Data_64_bytes[7];
	PlcInputs.ST50_4_DM260_Result_Data_64_bytes[8] := HwInputs.ST50_4_DM260_Result_Data_64_bytes[8];
	PlcInputs.ST50_4_DM260_Result_Data_64_bytes[9] := HwInputs.ST50_4_DM260_Result_Data_64_bytes[9];
	PlcInputs.ST50_4_DM260_Result_Data_64_bytes[10] := HwInputs.ST50_4_DM260_Result_Data_64_bytes[10];
	PlcInputs.ST50_4_DM260_Result_Data_64_bytes[11] := HwInputs.ST50_4_DM260_Result_Data_64_bytes[11];
	PlcInputs.ST50_4_DM260_Result_Data_64_bytes[12] := HwInputs.ST50_4_DM260_Result_Data_64_bytes[12];
	PlcInputs.ST50_4_DM260_Result_Data_64_bytes[13] := HwInputs.ST50_4_DM260_Result_Data_64_bytes[13];
	PlcInputs.ST50_4_DM260_Result_Data_64_bytes[14] := HwInputs.ST50_4_DM260_Result_Data_64_bytes[14];
	PlcInputs.ST50_4_DM260_Result_Data_64_bytes[15] := HwInputs.ST50_4_DM260_Result_Data_64_bytes[15];
	PlcInputs.ST50_4_DM260_Result_Data_64_bytes[16] := HwInputs.ST50_4_DM260_Result_Data_64_bytes[16];
	PlcInputs.ST50_4_DM260_Result_Data_64_bytes[17] := HwInputs.ST50_4_DM260_Result_Data_64_bytes[17];
	PlcInputs.ST50_4_DM260_Result_Data_64_bytes[18] := HwInputs.ST50_4_DM260_Result_Data_64_bytes[18];
	PlcInputs.ST50_4_DM260_Result_Data_64_bytes[19] := HwInputs.ST50_4_DM260_Result_Data_64_bytes[19];
	PlcInputs.ST50_4_DM260_Result_Data_64_bytes[20] := HwInputs.ST50_4_DM260_Result_Data_64_bytes[20];
	PlcInputs.ST50_4_DM260_Result_Data_64_bytes[21] := HwInputs.ST50_4_DM260_Result_Data_64_bytes[21];
	PlcInputs.ST50_4_DM260_Result_Data_64_bytes[22] := HwInputs.ST50_4_DM260_Result_Data_64_bytes[22];
	PlcInputs.ST50_4_DM260_Result_Data_64_bytes[23] := HwInputs.ST50_4_DM260_Result_Data_64_bytes[23];
	PlcInputs.ST50_4_DM260_Result_Data_64_bytes[24] := HwInputs.ST50_4_DM260_Result_Data_64_bytes[24];
	PlcInputs.ST50_4_DM260_Result_Data_64_bytes[25] := HwInputs.ST50_4_DM260_Result_Data_64_bytes[25];
	PlcInputs.ST50_4_DM260_Result_Data_64_bytes[26] := HwInputs.ST50_4_DM260_Result_Data_64_bytes[26];
	PlcInputs.ST50_4_DM260_Result_Data_64_bytes[27] := HwInputs.ST50_4_DM260_Result_Data_64_bytes[27];
	PlcInputs.ST50_4_DM260_Result_Data_64_bytes[28] := HwInputs.ST50_4_DM260_Result_Data_64_bytes[28];
	PlcInputs.ST50_4_DM260_Result_Data_64_bytes[29] := HwInputs.ST50_4_DM260_Result_Data_64_bytes[29];
	PlcInputs.ST50_4_DM260_Result_Data_64_bytes[30] := HwInputs.ST50_4_DM260_Result_Data_64_bytes[30];
	PlcInputs.ST50_4_DM260_Result_Data_64_bytes[31] := HwInputs.ST50_4_DM260_Result_Data_64_bytes[31];
	PlcInputs.ST50_4_DM260_Result_Data_64_bytes[32] := HwInputs.ST50_4_DM260_Result_Data_64_bytes[32];
	PlcInputs.ST50_4_DM260_Result_Data_64_bytes[33] := HwInputs.ST50_4_DM260_Result_Data_64_bytes[33];
	PlcInputs.ST50_4_DM260_Result_Data_64_bytes[34] := HwInputs.ST50_4_DM260_Result_Data_64_bytes[34];
	PlcInputs.ST50_4_DM260_Result_Data_64_bytes[35] := HwInputs.ST50_4_DM260_Result_Data_64_bytes[35];
	PlcInputs.ST50_4_DM260_Result_Data_64_bytes[36] := HwInputs.ST50_4_DM260_Result_Data_64_bytes[36];
	PlcInputs.ST50_4_DM260_Result_Data_64_bytes[37] := HwInputs.ST50_4_DM260_Result_Data_64_bytes[37];
	PlcInputs.ST50_4_DM260_Result_Data_64_bytes[38] := HwInputs.ST50_4_DM260_Result_Data_64_bytes[38];
	PlcInputs.ST50_4_DM260_Result_Data_64_bytes[39] := HwInputs.ST50_4_DM260_Result_Data_64_bytes[39];
	PlcInputs.ST50_4_DM260_Result_Data_64_bytes[40] := HwInputs.ST50_4_DM260_Result_Data_64_bytes[40];
	PlcInputs.ST50_4_DM260_Result_Data_64_bytes[41] := HwInputs.ST50_4_DM260_Result_Data_64_bytes[41];
	PlcInputs.ST50_4_DM260_Result_Data_64_bytes[42] := HwInputs.ST50_4_DM260_Result_Data_64_bytes[42];
	PlcInputs.ST50_4_DM260_Result_Data_64_bytes[43] := HwInputs.ST50_4_DM260_Result_Data_64_bytes[43];
	PlcInputs.ST50_4_DM260_Result_Data_64_bytes[44] := HwInputs.ST50_4_DM260_Result_Data_64_bytes[44];
	PlcInputs.ST50_4_DM260_Result_Data_64_bytes[45] := HwInputs.ST50_4_DM260_Result_Data_64_bytes[45];
	PlcInputs.ST50_4_DM260_Result_Data_64_bytes[46] := HwInputs.ST50_4_DM260_Result_Data_64_bytes[46];
	PlcInputs.ST50_4_DM260_Result_Data_64_bytes[47] := HwInputs.ST50_4_DM260_Result_Data_64_bytes[47];
	PlcInputs.ST50_4_DM260_Result_Data_64_bytes[48] := HwInputs.ST50_4_DM260_Result_Data_64_bytes[48];
	PlcInputs.ST50_4_DM260_Result_Data_64_bytes[49] := HwInputs.ST50_4_DM260_Result_Data_64_bytes[49];
	PlcInputs.ST50_4_DM260_Result_Data_64_bytes[50] := HwInputs.ST50_4_DM260_Result_Data_64_bytes[50];
	PlcInputs.ST50_4_DM260_Result_Data_64_bytes[51] := HwInputs.ST50_4_DM260_Result_Data_64_bytes[51];
	PlcInputs.ST50_4_DM260_Result_Data_64_bytes[52] := HwInputs.ST50_4_DM260_Result_Data_64_bytes[52];
	PlcInputs.ST50_4_DM260_Result_Data_64_bytes[53] := HwInputs.ST50_4_DM260_Result_Data_64_bytes[53];
	PlcInputs.ST50_4_DM260_Result_Data_64_bytes[54] := HwInputs.ST50_4_DM260_Result_Data_64_bytes[54];
	PlcInputs.ST50_4_DM260_Result_Data_64_bytes[55] := HwInputs.ST50_4_DM260_Result_Data_64_bytes[55];
	PlcInputs.ST50_4_DM260_Result_Data_64_bytes[56] := HwInputs.ST50_4_DM260_Result_Data_64_bytes[56];
	PlcInputs.ST50_4_DM260_Result_Data_64_bytes[57] := HwInputs.ST50_4_DM260_Result_Data_64_bytes[57];
	PlcInputs.ST50_4_DM260_Result_Data_64_bytes[58] := HwInputs.ST50_4_DM260_Result_Data_64_bytes[58];
	PlcInputs.ST50_4_DM260_Result_Data_64_bytes[59] := HwInputs.ST50_4_DM260_Result_Data_64_bytes[59];
	PlcInputs.ST50_4_DM260_Result_Data_64_bytes[60] := HwInputs.ST50_4_DM260_Result_Data_64_bytes[60];
	PlcInputs.ST50_4_DM260_Result_Data_64_bytes[61] := HwInputs.ST50_4_DM260_Result_Data_64_bytes[61];
	PlcInputs.ST50_4_DM260_Result_Data_64_bytes[62] := HwInputs.ST50_4_DM260_Result_Data_64_bytes[62];
	PlcInputs.ST50_4_DM260_Result_Data_64_bytes[63] := HwInputs.ST50_4_DM260_Result_Data_64_bytes[63];
	PlcInputs.ST50_4_DM260_Result_Data_64_bytes[64] := HwInputs.ST50_4_DM260_Result_Data_64_bytes[64];
	PlcInputs.ST50_4_DM260_Result_Data_64_bytes[65] := HwInputs.ST50_4_DM260_Result_Data_64_bytes[65];
	PlcInputs.ST50_4_DM260_Result_Data_64_bytes[66] := HwInputs.ST50_4_DM260_Result_Data_64_bytes[66];
	PlcInputs.ST50_4_DM260_Result_Data_64_bytes[67] := HwInputs.ST50_4_DM260_Result_Data_64_bytes[67];
	PlcInputs.ST50_4_DM260_Result_Data_64_bytes[68] := HwInputs.ST50_4_DM260_Result_Data_64_bytes[68];
	PlcInputs.ST50_4_DM260_Result_Data_64_bytes[69] := HwInputs.ST50_4_DM260_Result_Data_64_bytes[69];
	PlcInputs.ST50_4_DM260_Result_Data_64_bytes[70] := HwInputs.ST50_4_DM260_Result_Data_64_bytes[70];
	PlcInputs.ST50_4_DM260_Result_Data_64_bytes[71] := HwInputs.ST50_4_DM260_Result_Data_64_bytes[71];
END_FUNCTION
